// Mitsubishi GX Works2 project: RY300S2_3-4 24.07.21   PLC: Q03UDV
// RY300S2_3-4 24.07.21

PROGRAM MAIN
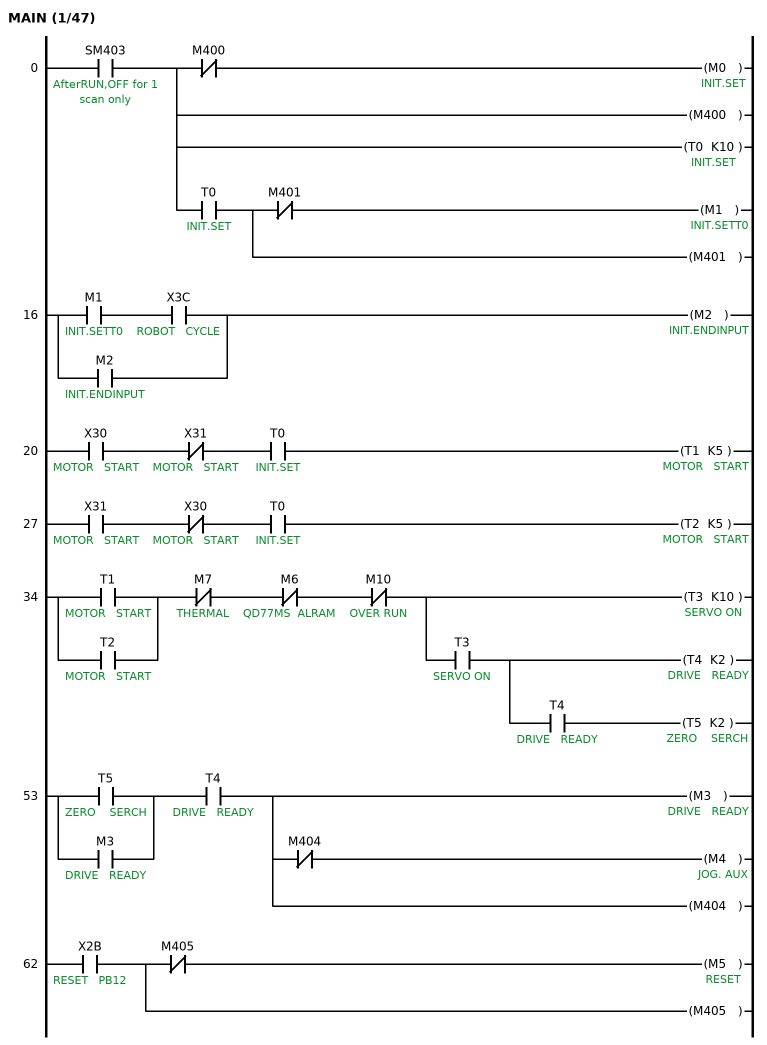
0     LD      SM403  ; AfterRUN,OFF for 1 scan only
      MPS
      ANI     M400
      OUT     M0  ; INIT.SET
      MPP
      OUT     M400
      OUT     T0 K10  ; INIT.SET
      AND     T0  ; INIT.SET
      MPS
      ANI     M401
      OUT     M1  ; INIT.SETT0
      MPP
      OUT     M401
16    LD      M1  ; INIT.SETT0
      AND     X3C  ; ROBOT   CYCLE
      OR      M2  ; INIT.ENDINPUT
      OUT     M2  ; INIT.ENDINPUT
20    LD      X30  ; MOTOR   START
      ANI     X31  ; MOTOR   START
      AND     T0  ; INIT.SET
      OUT     T1 K5  ; MOTOR   START
27    LD      X31  ; MOTOR   START
      ANI     X30  ; MOTOR   START
      AND     T0  ; INIT.SET
      OUT     T2 K5  ; MOTOR   START
34    LD      T1  ; MOTOR   START
      OR      T2  ; MOTOR   START
      ANI     M7  ; THERMAL
      ANI     M6  ; QD77MS  ALRAM
      ANI     M10  ; OVER RUN
      OUT     T3 K10  ; SERVO ON
      AND     T3  ; SERVO ON
      OUT     T4 K2  ; DRIVE   READY
      AND     T4  ; DRIVE   READY
      OUT     T5 K2  ; ZERO    SERCH
53    LD      T5  ; ZERO    SERCH
      OR      M3  ; DRIVE   READY
      AND     T4  ; DRIVE   READY
      OUT     M3  ; DRIVE   READY
      MPS
      ANI     M404
      OUT     M4  ; JOG. AUX
      MPP
      OUT     M404
62    LD      X2B  ; RESET   PB12
      MPS
      ANI     M405
      OUT     M5  ; RESET
      MPP
      OUT     M405
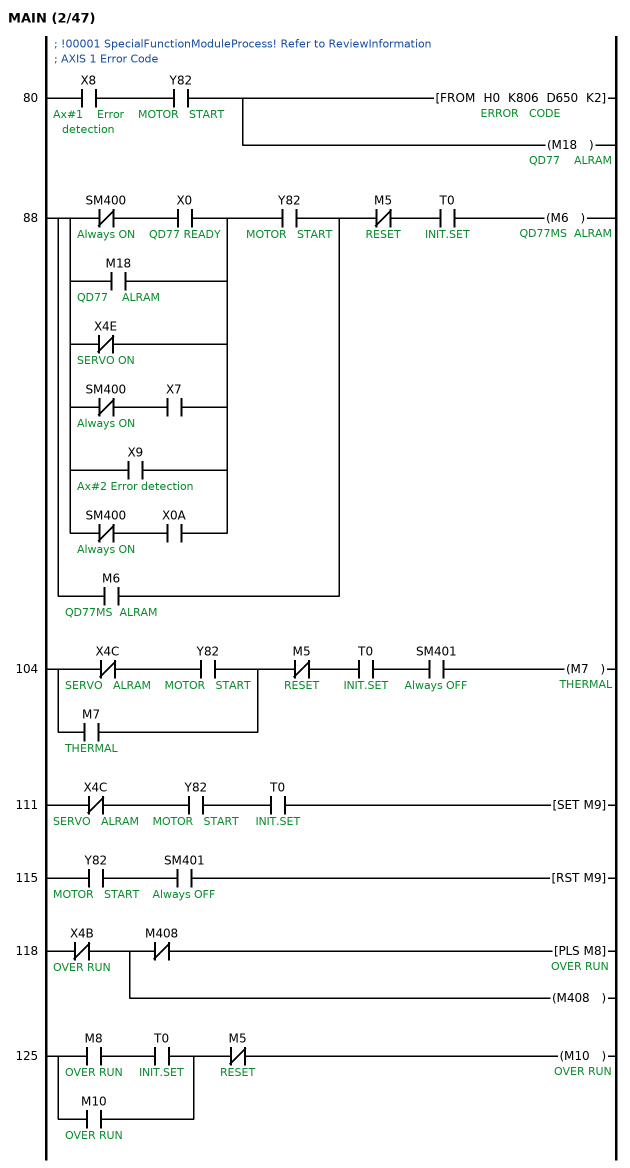
; !00001 SpecialFunctionModuleProcess! Refer to ReviewInformation
; AXIS 1 Error Code
80    LD      X8  ; Ax#1    Error   detection
      AND     Y82  ; MOTOR   START
      FROM    H0 K806 D650 K2  ; ERROR   CODE
      OUT     M18  ; QD77    ALRAM
88    LDI     SM400  ; Always ON
      AND     X0  ; QD77 READY
      OR      M18  ; QD77    ALRAM
      ORI     X4E  ; SERVO ON
      LDI     SM400  ; Always ON
      AND     X7
      ORB
      OR      X9  ; Ax#2 Error detection
      LDI     SM400  ; Always ON
      AND     X0A
      ORB
      AND     Y82  ; MOTOR   START
      OR      M6  ; QD77MS  ALRAM
      ANI     M5  ; RESET
      AND     T0  ; INIT.SET
      OUT     M6  ; QD77MS  ALRAM
104   LDI     X4C  ; SERVO   ALRAM
      AND     Y82  ; MOTOR   START
      OR      M7  ; THERMAL
      ANI     M5  ; RESET
      AND     T0  ; INIT.SET
      AND     SM401  ; Always OFF
      OUT     M7  ; THERMAL
111   LDI     X4C  ; SERVO   ALRAM
      AND     Y82  ; MOTOR   START
      AND     T0  ; INIT.SET
      SET     M9
115   LD      Y82  ; MOTOR   START
      AND     SM401  ; Always OFF
      RST     M9
118   LDI     X4B  ; OVER RUN
      MPS
      ANI     M408
      PLS     M8  ; OVER RUN
      MPP
      OUT     M408
125   LD      M8  ; OVER RUN
      AND     T0  ; INIT.SET
      OR      M10  ; OVER RUN
      ANI     M5  ; RESET
      OUT     M10  ; OVER RUN
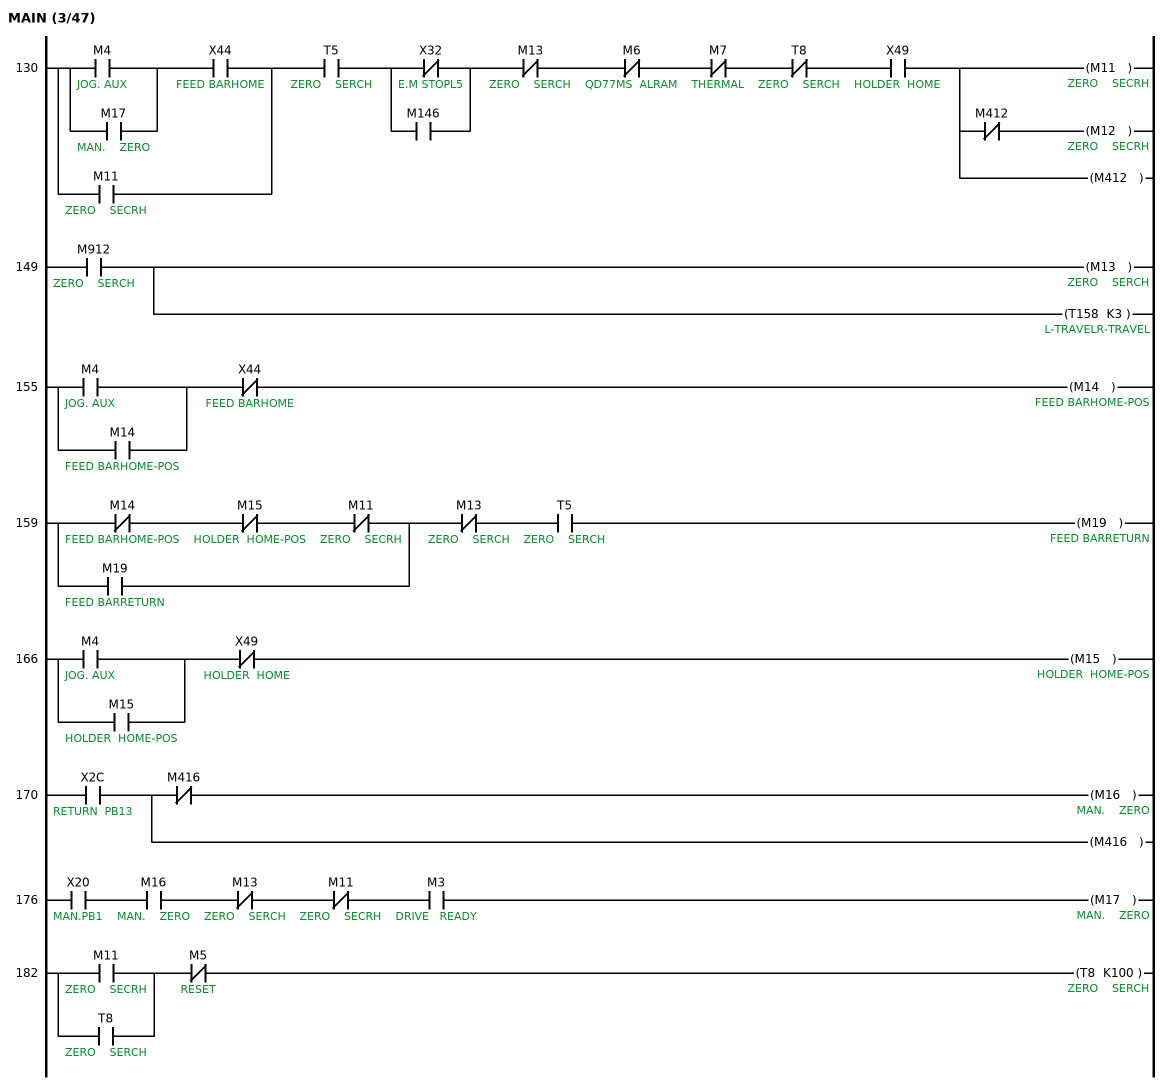
130   LD      M4  ; JOG. AUX
      OR      M17  ; MAN.    ZERO
      AND     X44  ; FEED BARHOME
      OR      M11  ; ZERO    SECRH
      AND     T5  ; ZERO    SERCH
      LDI     X32  ; E.M STOPL5
      OR      M146
      ANB
      ANI     M13  ; ZERO    SERCH
      ANI     M6  ; QD77MS  ALRAM
      ANI     M7  ; THERMAL
      ANI     T8  ; ZERO    SERCH
      AND     X49  ; HOLDER  HOME
      OUT     M11  ; ZERO    SECRH
      MPS
      ANI     M412
      OUT     M12  ; ZERO    SECRH
      MPP
      OUT     M412
149   LD      M912  ; ZERO    SERCH
      OUT     M13  ; ZERO    SERCH
      OUT     T158 K3  ; L-TRAVELR-TRAVEL
155   LD      M4  ; JOG. AUX
      OR      M14  ; FEED BARHOME-POS
      ANI     X44  ; FEED BARHOME
      OUT     M14  ; FEED BARHOME-POS
159   LDI     M14  ; FEED BARHOME-POS
      ANI     M15  ; HOLDER  HOME-POS
      ANI     M11  ; ZERO    SECRH
      OR      M19  ; FEED BARRETURN
      ANI     M13  ; ZERO    SERCH
      AND     T5  ; ZERO    SERCH
      OUT     M19  ; FEED BARRETURN
166   LD      M4  ; JOG. AUX
      OR      M15  ; HOLDER  HOME-POS
      ANI     X49  ; HOLDER  HOME
      OUT     M15  ; HOLDER  HOME-POS
170   LD      X2C  ; RETURN  PB13
      MPS
      ANI     M416
      OUT     M16  ; MAN.    ZERO
      MPP
      OUT     M416
176   LD      X20  ; MAN.PB1
      AND     M16  ; MAN.    ZERO
      ANI     M13  ; ZERO    SERCH
      ANI     M11  ; ZERO    SECRH
      AND     M3  ; DRIVE   READY
      OUT     M17  ; MAN.    ZERO
182   LD      M11  ; ZERO    SECRH
      OR      T8  ; ZERO    SERCH
      ANI     M5  ; RESET
      OUT     T8 K100  ; ZERO    SERCH
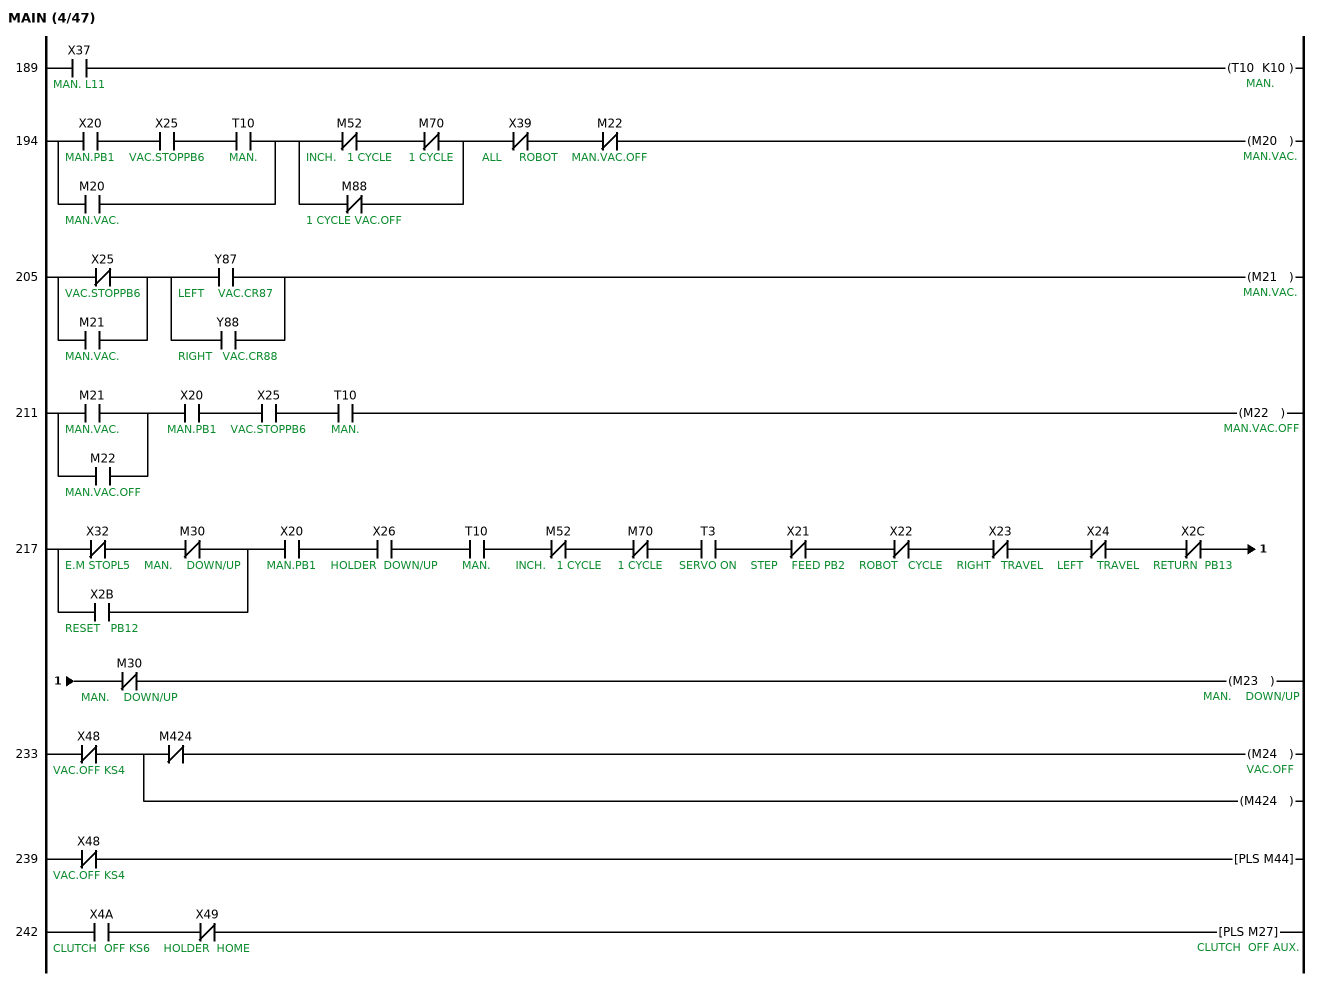
189   LD      X37  ; MAN. L11
      OUT     T10 K10  ; MAN.
194   LD      X20  ; MAN.PB1
      AND     X25  ; VAC.STOPPB6
      AND     T10  ; MAN.
      OR      M20  ; MAN.VAC.
      LDI     M52  ; INCH.   1 CYCLE
      ANI     M70  ; 1 CYCLE
      ORI     M88  ; 1 CYCLE VAC.OFF
      ANB
      ANI     X39  ; ALL     ROBOT
      ANI     M22  ; MAN.VAC.OFF
      OUT     M20  ; MAN.VAC.
205   LDI     X25  ; VAC.STOPPB6
      OR      M21  ; MAN.VAC.
      LD      Y87  ; LEFT    VAC.CR87
      OR      Y88  ; RIGHT   VAC.CR88
      ANB
      OUT     M21  ; MAN.VAC.
211   LD      M21  ; MAN.VAC.
      OR      M22  ; MAN.VAC.OFF
      AND     X20  ; MAN.PB1
      AND     X25  ; VAC.STOPPB6
      AND     T10  ; MAN.
      OUT     M22  ; MAN.VAC.OFF
217   LDI     X32  ; E.M STOPL5
      ANI     M30  ; MAN.    DOWN/UP
      OR      X2B  ; RESET   PB12
      AND     X20  ; MAN.PB1
      AND     X26  ; HOLDER  DOWN/UP
      AND     T10  ; MAN.
      ANI     M52  ; INCH.   1 CYCLE
      ANI     M70  ; 1 CYCLE
      AND     T3  ; SERVO ON
      ANI     X21  ; STEP    FEED PB2
      ANI     X22  ; ROBOT   CYCLE
      ANI     X23  ; RIGHT   TRAVEL
      ANI     X24  ; LEFT    TRAVEL
      ANI     X2C  ; RETURN  PB13
      ANI     M30  ; MAN.    DOWN/UP
      OUT     M23  ; MAN.    DOWN/UP
233   LDI     X48  ; VAC.OFF KS4
      MPS
      ANI     M424
      OUT     M24  ; VAC.OFF
      MPP
      OUT     M424
239   LDI     X48  ; VAC.OFF KS4
      PLS     M44
242   LD      X4A  ; CLUTCH  OFF KS6
      ANI     X49  ; HOLDER  HOME
      PLS     M27  ; CLUTCH  OFF AUX.
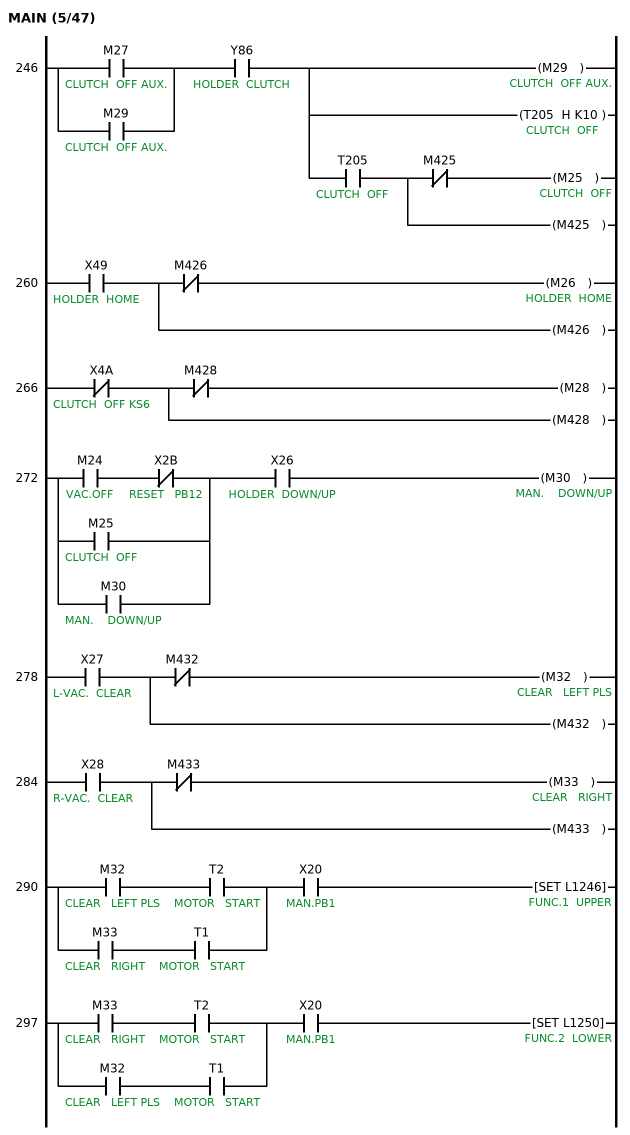
246   LD      M27  ; CLUTCH  OFF AUX.
      OR      M29  ; CLUTCH  OFF AUX.
      AND     Y86  ; HOLDER  CLUTCH
      OUT     M29  ; CLUTCH  OFF AUX.
      OUTH    T205 K10  ; CLUTCH  OFF
      AND     T205  ; CLUTCH  OFF
      MPS
      ANI     M425
      OUT     M25  ; CLUTCH  OFF
      MPP
      OUT     M425
260   LD      X49  ; HOLDER  HOME
      MPS
      ANI     M426
      OUT     M26  ; HOLDER  HOME
      MPP
      OUT     M426
266   LDI     X4A  ; CLUTCH  OFF KS6
      MPS
      ANI     M428
      OUT     M28
      MPP
      OUT     M428
272   LD      M24  ; VAC.OFF
      ANI     X2B  ; RESET   PB12
      OR      M25  ; CLUTCH  OFF
      OR      M30  ; MAN.    DOWN/UP
      AND     X26  ; HOLDER  DOWN/UP
      OUT     M30  ; MAN.    DOWN/UP
278   LD      X27  ; L-VAC.  CLEAR
      MPS
      ANI     M432
      OUT     M32  ; CLEAR   LEFT PLS
      MPP
      OUT     M432
284   LD      X28  ; R-VAC.  CLEAR
      MPS
      ANI     M433
      OUT     M33  ; CLEAR   RIGHT
      MPP
      OUT     M433
290   LD      M32  ; CLEAR   LEFT PLS
      AND     T2  ; MOTOR   START
      LD      M33  ; CLEAR   RIGHT
      AND     T1  ; MOTOR   START
      ORB
      AND     X20  ; MAN.PB1
      SET     L1246  ; FUNC.1  UPPER
297   LD      M33  ; CLEAR   RIGHT
      AND     T2  ; MOTOR   START
      LD      M32  ; CLEAR   LEFT PLS
      AND     T1  ; MOTOR   START
      ORB
      AND     X20  ; MAN.PB1
      SET     L1250  ; FUNC.2  LOWER
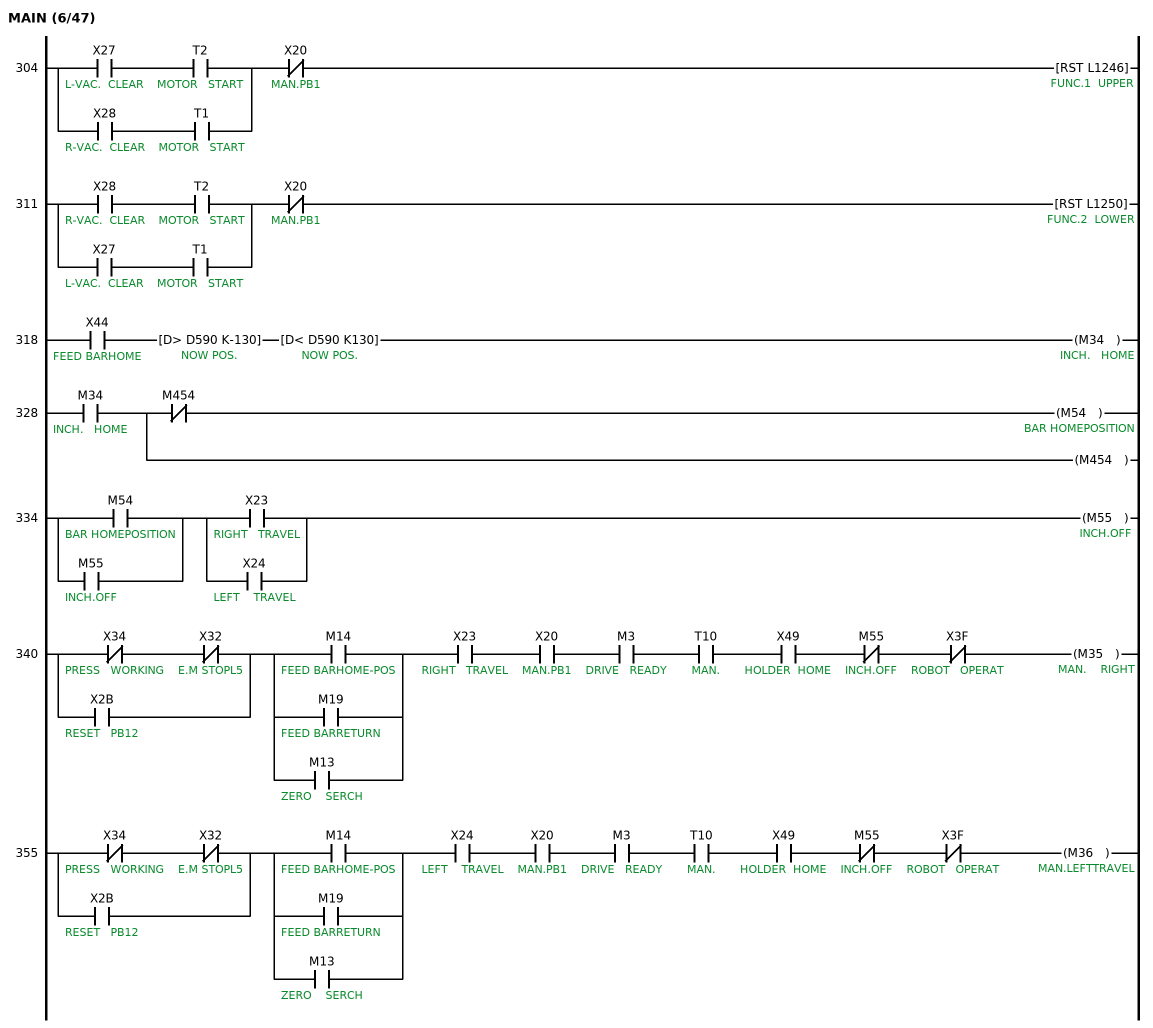
304   LD      X27  ; L-VAC.  CLEAR
      AND     T2  ; MOTOR   START
      LD      X28  ; R-VAC.  CLEAR
      AND     T1  ; MOTOR   START
      ORB
      ANI     X20  ; MAN.PB1
      RST     L1246  ; FUNC.1  UPPER
311   LD      X28  ; R-VAC.  CLEAR
      AND     T2  ; MOTOR   START
      LD      X27  ; L-VAC.  CLEAR
      AND     T1  ; MOTOR   START
      ORB
      ANI     X20  ; MAN.PB1
      RST     L1250  ; FUNC.2  LOWER
318   LD      X44  ; FEED BARHOME
      ANDD>   D590 K-130  ; NOW POS.
      ANDD<   D590 K130  ; NOW POS.
      OUT     M34  ; INCH.   HOME
328   LD      M34  ; INCH.   HOME
      MPS
      ANI     M454
      OUT     M54  ; BAR HOMEPOSITION
      MPP
      OUT     M454
334   LD      M54  ; BAR HOMEPOSITION
      OR      M55  ; INCH.OFF
      LD      X23  ; RIGHT   TRAVEL
      OR      X24  ; LEFT    TRAVEL
      ANB
      OUT     M55  ; INCH.OFF
340   LDI     X34  ; PRESS   WORKING
      ANI     X32  ; E.M STOPL5
      OR      X2B  ; RESET   PB12
      LD      M14  ; FEED BARHOME-POS
      OR      M19  ; FEED BARRETURN
      OR      M13  ; ZERO    SERCH
      ANB
      AND     X23  ; RIGHT   TRAVEL
      AND     X20  ; MAN.PB1
      AND     M3  ; DRIVE   READY
      AND     T10  ; MAN.
      AND     X49  ; HOLDER  HOME
      ANI     M55  ; INCH.OFF
      ANI     X3F  ; ROBOT   OPERAT
      OUT     M35  ; MAN.    RIGHT
355   LDI     X34  ; PRESS   WORKING
      ANI     X32  ; E.M STOPL5
      OR      X2B  ; RESET   PB12
      LD      M14  ; FEED BARHOME-POS
      OR      M19  ; FEED BARRETURN
      OR      M13  ; ZERO    SERCH
      ANB
      AND     X24  ; LEFT    TRAVEL
      AND     X20  ; MAN.PB1
      AND     M3  ; DRIVE   READY
      AND     T10  ; MAN.
      AND     X49  ; HOLDER  HOME
      ANI     M55  ; INCH.OFF
      ANI     X3F  ; ROBOT   OPERAT
      OUT     M36  ; MAN.LEFTTRAVEL
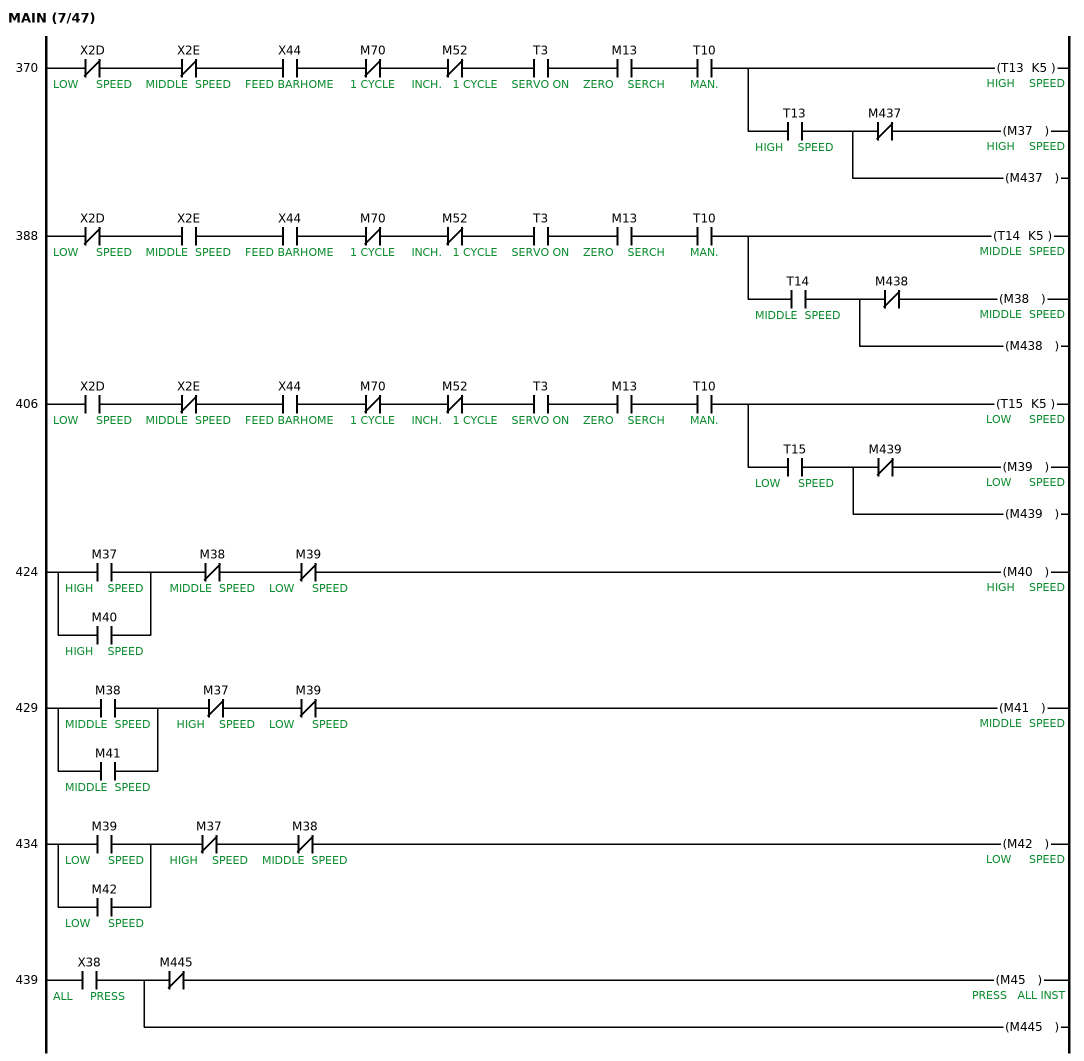
370   LDI     X2D  ; LOW     SPEED
      ANI     X2E  ; MIDDLE  SPEED
      AND     X44  ; FEED BARHOME
      ANI     M70  ; 1 CYCLE
      ANI     M52  ; INCH.   1 CYCLE
      AND     T3  ; SERVO ON
      AND     M13  ; ZERO    SERCH
      AND     T10  ; MAN.
      OUT     T13 K5  ; HIGH    SPEED
      AND     T13  ; HIGH    SPEED
      MPS
      ANI     M437
      OUT     M37  ; HIGH    SPEED
      MPP
      OUT     M437
388   LDI     X2D  ; LOW     SPEED
      AND     X2E  ; MIDDLE  SPEED
      AND     X44  ; FEED BARHOME
      ANI     M70  ; 1 CYCLE
      ANI     M52  ; INCH.   1 CYCLE
      AND     T3  ; SERVO ON
      AND     M13  ; ZERO    SERCH
      AND     T10  ; MAN.
      OUT     T14 K5  ; MIDDLE  SPEED
      AND     T14  ; MIDDLE  SPEED
      MPS
      ANI     M438
      OUT     M38  ; MIDDLE  SPEED
      MPP
      OUT     M438
406   LD      X2D  ; LOW     SPEED
      ANI     X2E  ; MIDDLE  SPEED
      AND     X44  ; FEED BARHOME
      ANI     M70  ; 1 CYCLE
      ANI     M52  ; INCH.   1 CYCLE
      AND     T3  ; SERVO ON
      AND     M13  ; ZERO    SERCH
      AND     T10  ; MAN.
      OUT     T15 K5  ; LOW     SPEED
      AND     T15  ; LOW     SPEED
      MPS
      ANI     M439
      OUT     M39  ; LOW     SPEED
      MPP
      OUT     M439
424   LD      M37  ; HIGH    SPEED
      OR      M40  ; HIGH    SPEED
      ANI     M38  ; MIDDLE  SPEED
      ANI     M39  ; LOW     SPEED
      OUT     M40  ; HIGH    SPEED
429   LD      M38  ; MIDDLE  SPEED
      OR      M41  ; MIDDLE  SPEED
      ANI     M37  ; HIGH    SPEED
      ANI     M39  ; LOW     SPEED
      OUT     M41  ; MIDDLE  SPEED
434   LD      M39  ; LOW     SPEED
      OR      M42  ; LOW     SPEED
      ANI     M37  ; HIGH    SPEED
      ANI     M38  ; MIDDLE  SPEED
      OUT     M42  ; LOW     SPEED
439   LD      X38  ; ALL     PRESS
      MPS
      ANI     M445
      OUT     M45  ; PRESS   ALL INST
      MPP
      OUT     M445
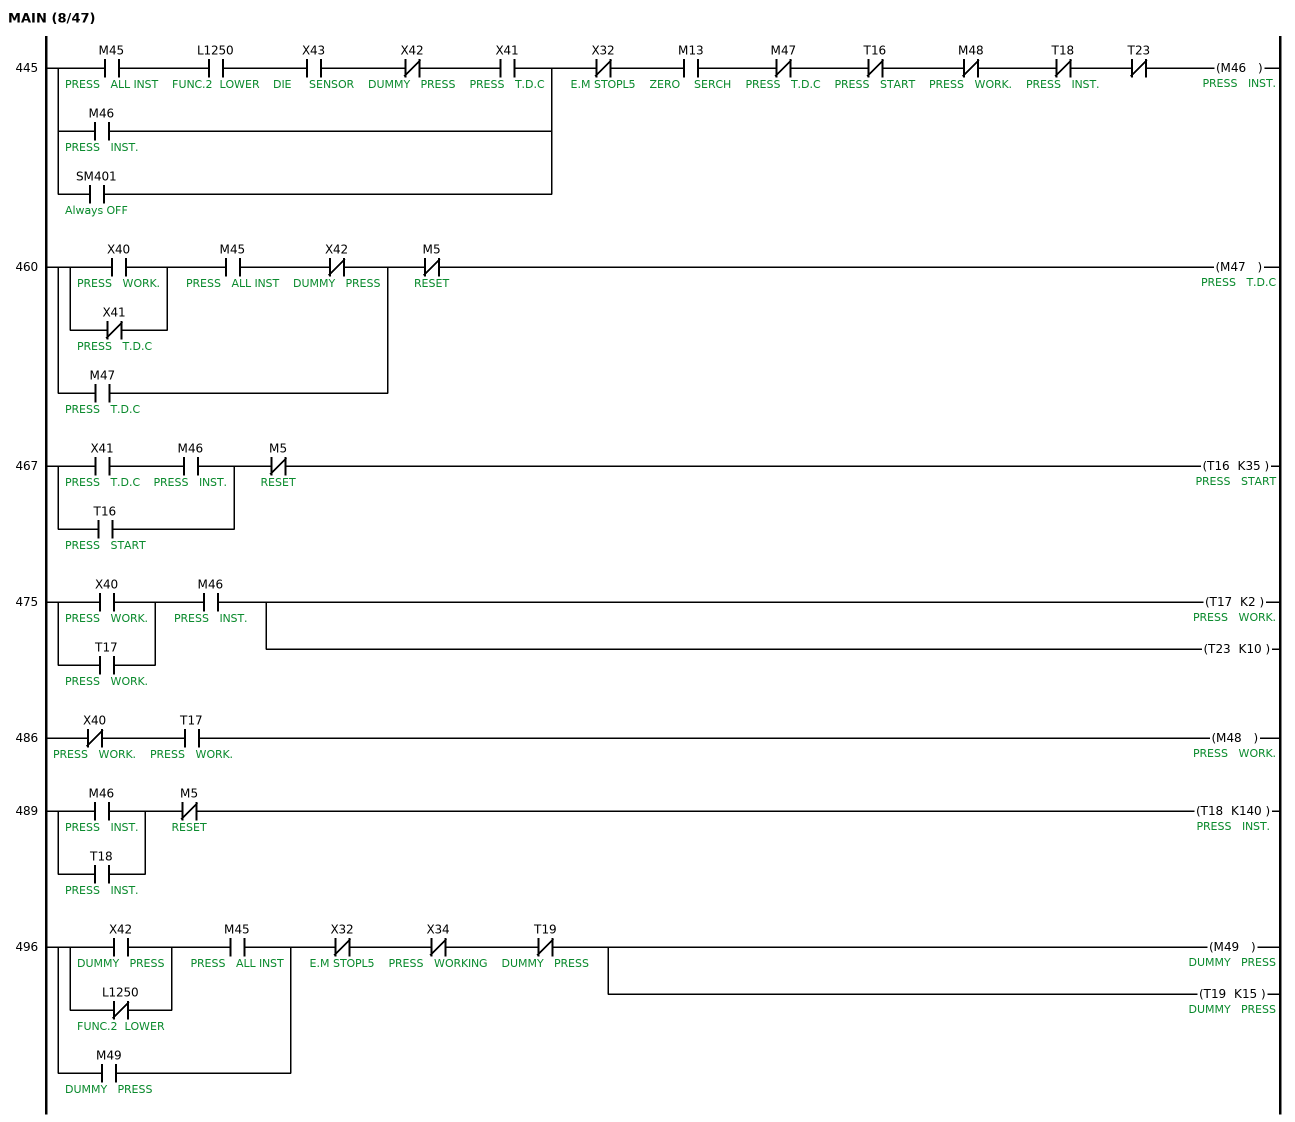
445   LD      M45  ; PRESS   ALL INST
      AND     L1250  ; FUNC.2  LOWER
      AND     X43  ; DIE     SENSOR
      ANI     X42  ; DUMMY   PRESS
      AND     X41  ; PRESS   T.D.C
      OR      M46  ; PRESS   INST.
      OR      SM401  ; Always OFF
      ANI     X32  ; E.M STOPL5
      AND     M13  ; ZERO    SERCH
      ANI     M47  ; PRESS   T.D.C
      ANI     T16  ; PRESS   START
      ANI     M48  ; PRESS   WORK.
      ANI     T18  ; PRESS   INST.
      ANI     T23
      OUT     M46  ; PRESS   INST.
460   LD      X40  ; PRESS   WORK.
      ORI     X41  ; PRESS   T.D.C
      AND     M45  ; PRESS   ALL INST
      ANI     X42  ; DUMMY   PRESS
      OR      M47  ; PRESS   T.D.C
      ANI     M5  ; RESET
      OUT     M47  ; PRESS   T.D.C
467   LD      X41  ; PRESS   T.D.C
      AND     M46  ; PRESS   INST.
      OR      T16  ; PRESS   START
      ANI     M5  ; RESET
      OUT     T16 K35  ; PRESS   START
475   LD      X40  ; PRESS   WORK.
      OR      T17  ; PRESS   WORK.
      AND     M46  ; PRESS   INST.
      OUT     T17 K2  ; PRESS   WORK.
      OUT     T23 K10
486   LDI     X40  ; PRESS   WORK.
      AND     T17  ; PRESS   WORK.
      OUT     M48  ; PRESS   WORK.
489   LD      M46  ; PRESS   INST.
      OR      T18  ; PRESS   INST.
      ANI     M5  ; RESET
      OUT     T18 K140  ; PRESS   INST.
496   LD      X42  ; DUMMY   PRESS
      ORI     L1250  ; FUNC.2  LOWER
      AND     M45  ; PRESS   ALL INST
      OR      M49  ; DUMMY   PRESS
      ANI     X32  ; E.M STOPL5
      ANI     X34  ; PRESS   WORKING
      ANI     T19  ; DUMMY   PRESS
      OUT     M49  ; DUMMY   PRESS
      OUT     T19 K15  ; DUMMY   PRESS
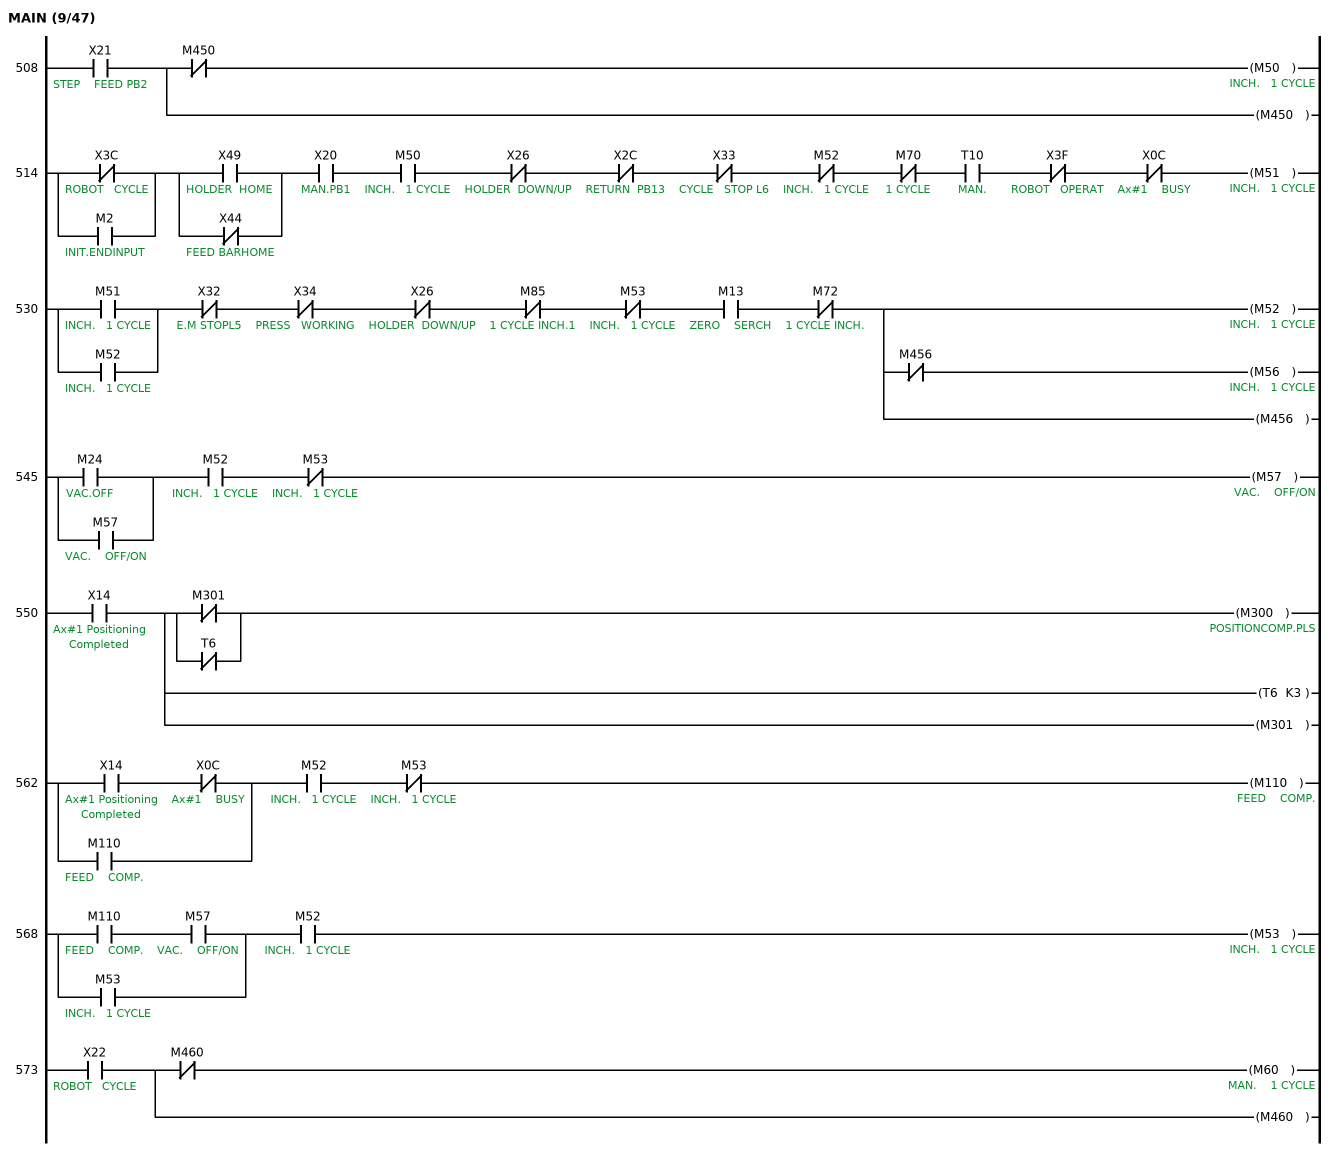
508   LD      X21  ; STEP    FEED PB2
      MPS
      ANI     M450
      OUT     M50  ; INCH.   1 CYCLE
      MPP
      OUT     M450
514   LDI     X3C  ; ROBOT   CYCLE
      OR      M2  ; INIT.ENDINPUT
      LD      X49  ; HOLDER  HOME
      ORI     X44  ; FEED BARHOME
      ANB
      AND     X20  ; MAN.PB1
      AND     M50  ; INCH.   1 CYCLE
      ANI     X26  ; HOLDER  DOWN/UP
      ANI     X2C  ; RETURN  PB13
      ANI     X33  ; CYCLE   STOP L6
      ANI     M52  ; INCH.   1 CYCLE
      ANI     M70  ; 1 CYCLE
      AND     T10  ; MAN.
      ANI     X3F  ; ROBOT   OPERAT
      ANI     X0C  ; Ax#1    BUSY
      OUT     M51  ; INCH.   1 CYCLE
530   LD      M51  ; INCH.   1 CYCLE
      OR      M52  ; INCH.   1 CYCLE
      ANI     X32  ; E.M STOPL5
      ANI     X34  ; PRESS   WORKING
      ANI     X26  ; HOLDER  DOWN/UP
      ANI     M85  ; 1 CYCLE INCH.1
      ANI     M53  ; INCH.   1 CYCLE
      AND     M13  ; ZERO    SERCH
      ANI     M72  ; 1 CYCLE INCH.
      OUT     M52  ; INCH.   1 CYCLE
      MPS
      ANI     M456
      OUT     M56  ; INCH.   1 CYCLE
      MPP
      OUT     M456
545   LD      M24  ; VAC.OFF
      OR      M57  ; VAC.    OFF/ON
      AND     M52  ; INCH.   1 CYCLE
      ANI     M53  ; INCH.   1 CYCLE
      OUT     M57  ; VAC.    OFF/ON
550   LD      X14  ; Ax#1 PositioningCompleted
      MPS
      LDI     M301
      ORI     T6
      ANB
      OUT     M300  ; POSITIONCOMP.PLS
      MPP
      OUT     T6 K3
      OUT     M301
562   LD      X14  ; Ax#1 PositioningCompleted
      ANI     X0C  ; Ax#1    BUSY
      OR      M110  ; FEED    COMP.
      AND     M52  ; INCH.   1 CYCLE
      ANI     M53  ; INCH.   1 CYCLE
      OUT     M110  ; FEED    COMP.
568   LD      M110  ; FEED    COMP.
      AND     M57  ; VAC.    OFF/ON
      OR      M53  ; INCH.   1 CYCLE
      AND     M52  ; INCH.   1 CYCLE
      OUT     M53  ; INCH.   1 CYCLE
573   LD      X22  ; ROBOT   CYCLE
      MPS
      ANI     M460
      OUT     M60  ; MAN.    1 CYCLE
      MPP
      OUT     M460
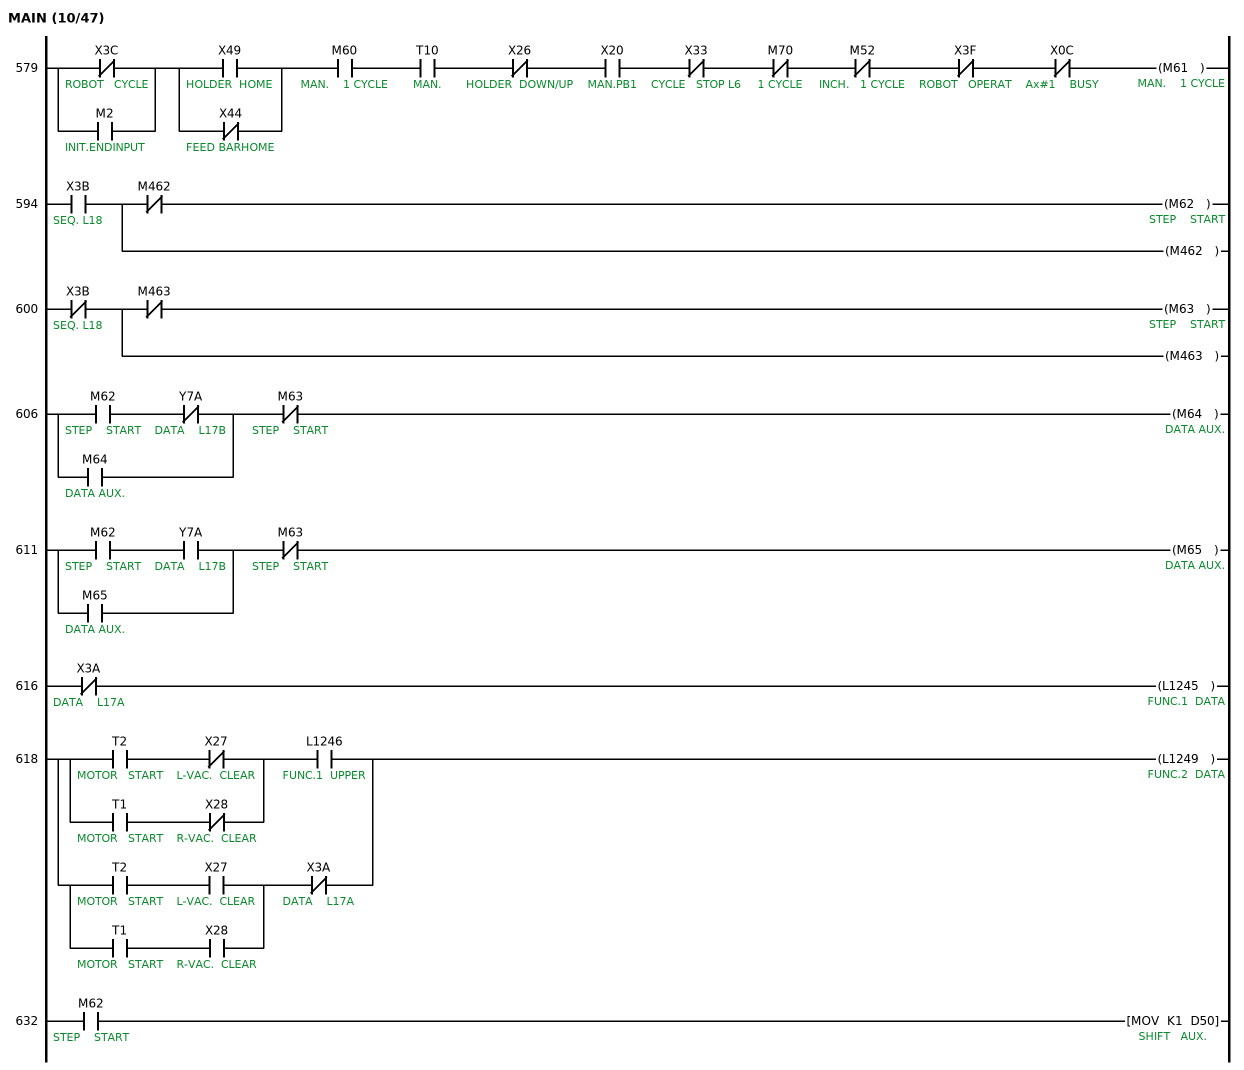
579   LDI     X3C  ; ROBOT   CYCLE
      OR      M2  ; INIT.ENDINPUT
      LD      X49  ; HOLDER  HOME
      ORI     X44  ; FEED BARHOME
      ANB
      AND     M60  ; MAN.    1 CYCLE
      AND     T10  ; MAN.
      ANI     X26  ; HOLDER  DOWN/UP
      AND     X20  ; MAN.PB1
      ANI     X33  ; CYCLE   STOP L6
      ANI     M70  ; 1 CYCLE
      ANI     M52  ; INCH.   1 CYCLE
      ANI     X3F  ; ROBOT   OPERAT
      ANI     X0C  ; Ax#1    BUSY
      OUT     M61  ; MAN.    1 CYCLE
594   LD      X3B  ; SEQ. L18
      MPS
      ANI     M462
      OUT     M62  ; STEP    START
      MPP
      OUT     M462
600   LDI     X3B  ; SEQ. L18
      MPS
      ANI     M463
      OUT     M63  ; STEP    START
      MPP
      OUT     M463
606   LD      M62  ; STEP    START
      ANI     Y7A  ; DATA    L17B
      OR      M64  ; DATA AUX.
      ANI     M63  ; STEP    START
      OUT     M64  ; DATA AUX.
611   LD      M62  ; STEP    START
      AND     Y7A  ; DATA    L17B
      OR      M65  ; DATA AUX.
      ANI     M63  ; STEP    START
      OUT     M65  ; DATA AUX.
616   LDI     X3A  ; DATA    L17A
      OUT     L1245  ; FUNC.1  DATA
618   LD      T2  ; MOTOR   START
      ANI     X27  ; L-VAC.  CLEAR
      LD      T1  ; MOTOR   START
      ANI     X28  ; R-VAC.  CLEAR
      ORB
      AND     L1246  ; FUNC.1  UPPER
      LD      T2  ; MOTOR   START
      AND     X27  ; L-VAC.  CLEAR
      LD      T1  ; MOTOR   START
      AND     X28  ; R-VAC.  CLEAR
      ORB
      ANI     X3A  ; DATA    L17A
      ORB
      OUT     L1249  ; FUNC.2  DATA
632   LD      M62  ; STEP    START
      MOV     K1 D50  ; SHIFT   AUX.
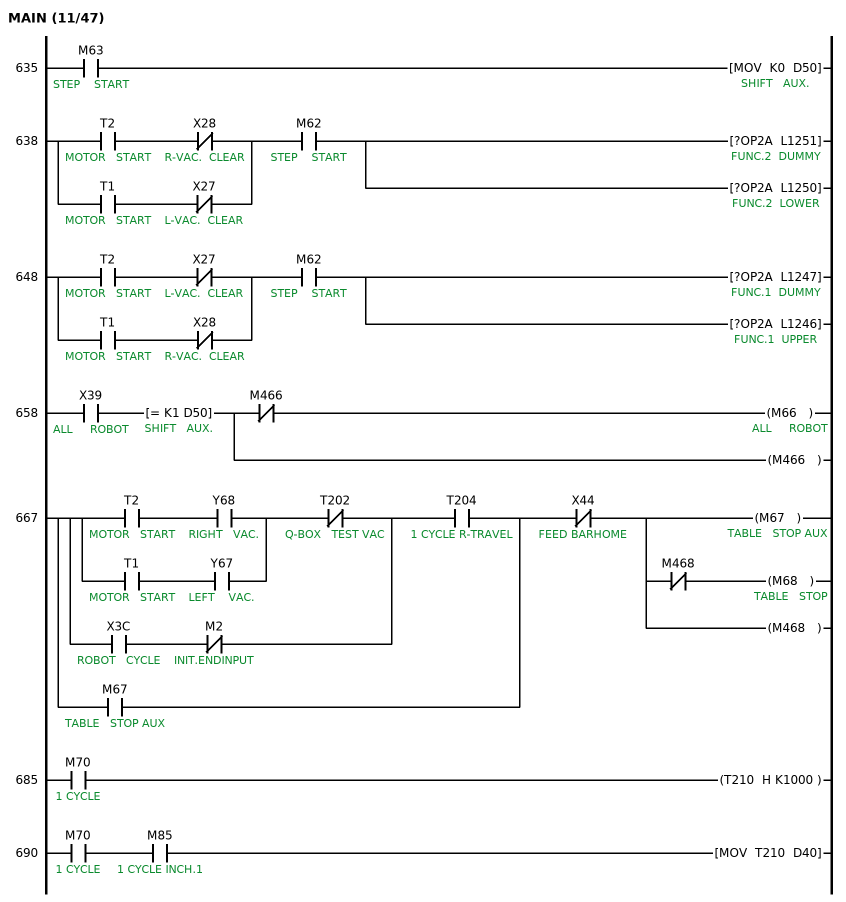
635   LD      M63  ; STEP    START
      MOV     K0 D50
638   LD      T2  ; MOTOR   START
      ANI     X28  ; R-VAC.  CLEAR
      LD      T1  ; MOTOR   START
      ANI     X27  ; L-VAC.  CLEAR
      ORB
      AND     M62  ; STEP    START
      ?OP2A   L1251  ; FUNC.2  DUMMY
      ?OP2A   L1250
648   LD      T2  ; MOTOR   START
      ANI     X27  ; L-VAC.  CLEAR
      LD      T1  ; MOTOR   START
      ANI     X28  ; R-VAC.  CLEAR
      ORB
      AND     M62  ; STEP    START
      ?OP2A   L1247  ; FUNC.1  DUMMY
      ?OP2A   L1246
658   LD      X39  ; ALL     ROBOT
      AND=    K1 D50  ; SHIFT   AUX.
      MPS
      ANI     M466
      OUT     M66  ; ALL     ROBOT
      MPP
      OUT     M466
667   LD      T2  ; MOTOR   START
      AND     Y68  ; RIGHT   VAC.
      LD      T1  ; MOTOR   START
      AND     Y67  ; LEFT    VAC.
      ORB
      ANI     T202  ; Q-BOX   TEST VAC
      LD      X3C  ; ROBOT   CYCLE
      ANI     M2  ; INIT.ENDINPUT
      ORB
      AND     T204  ; 1 CYCLE R-TRAVEL
      OR      M67  ; TABLE   STOP AUX
      ANI     X44  ; FEED BARHOME
      OUT     M67  ; TABLE   STOP AUX
      MPS
      ANI     M468
      OUT     M68  ; TABLE   STOP
      MPP
      OUT     M468
685   LD      M70  ; 1 CYCLE
      OUTH    T210 K1000
690   LD      M70  ; 1 CYCLE
      AND     M85  ; 1 CYCLE INCH.1
      MOV     T210 D40
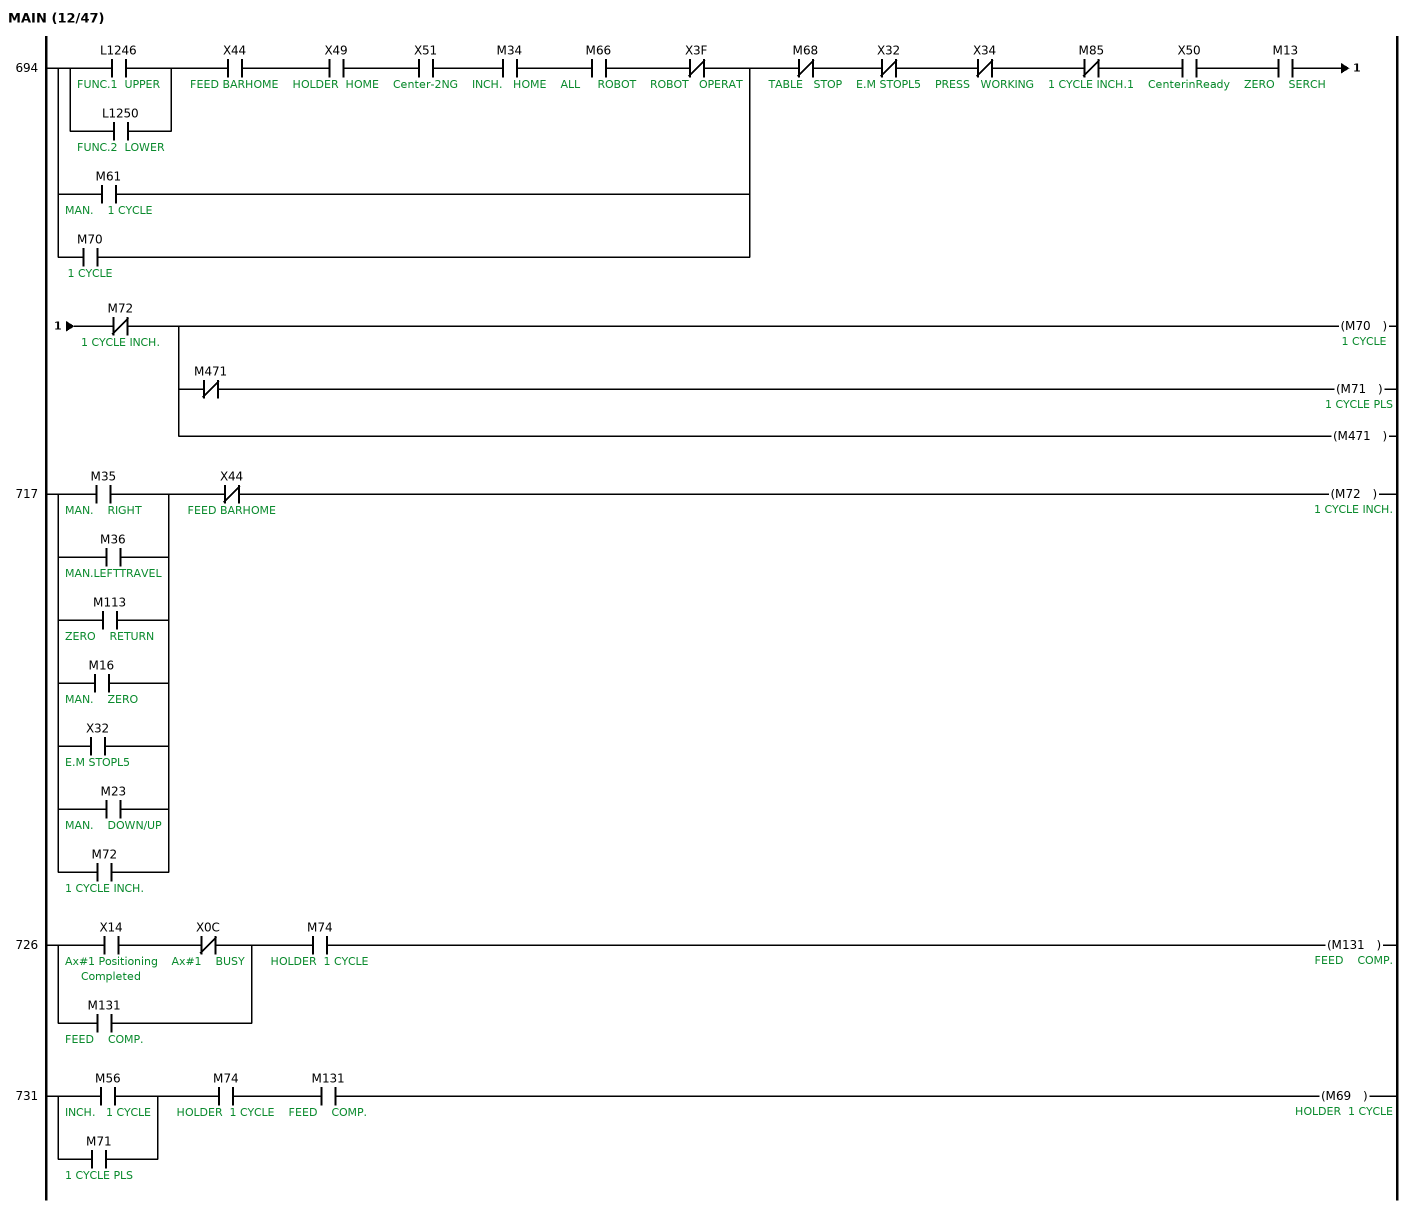
694   LD      L1246  ; FUNC.1  UPPER
      OR      L1250  ; FUNC.2  LOWER
      AND     X44  ; FEED BARHOME
      AND     X49  ; HOLDER  HOME
      AND     X51  ; Center-2NG
      AND     M34  ; INCH.   HOME
      AND     M66  ; ALL     ROBOT
      ANI     X3F  ; ROBOT   OPERAT
      OR      M61  ; MAN.    1 CYCLE
      OR      M70  ; 1 CYCLE
      ANI     M68  ; TABLE   STOP
      ANI     X32  ; E.M STOPL5
      ANI     X34  ; PRESS   WORKING
      ANI     M85  ; 1 CYCLE INCH.1
      AND     X50  ; CenterinReady
      AND     M13  ; ZERO    SERCH
      ANI     M72  ; 1 CYCLE INCH.
      OUT     M70  ; 1 CYCLE
      MPS
      ANI     M471
      OUT     M71  ; 1 CYCLE PLS
      MPP
      OUT     M471
717   LD      M35  ; MAN.    RIGHT
      OR      M36  ; MAN.LEFTTRAVEL
      OR      M113  ; ZERO    RETURN
      OR      M16  ; MAN.    ZERO
      OR      X32  ; E.M STOPL5
      OR      M23  ; MAN.    DOWN/UP
      OR      M72  ; 1 CYCLE INCH.
      ANI     X44  ; FEED BARHOME
      OUT     M72  ; 1 CYCLE INCH.
726   LD      X14  ; Ax#1 PositioningCompleted
      ANI     X0C  ; Ax#1    BUSY
      OR      M131  ; FEED    COMP.
      AND     M74  ; HOLDER  1 CYCLE
      OUT     M131  ; FEED    COMP.
731   LD      M56  ; INCH.   1 CYCLE
      OR      M71  ; 1 CYCLE PLS
      AND     M74  ; HOLDER  1 CYCLE
      AND     M131  ; FEED    COMP.
      OUT     M69  ; HOLDER  1 CYCLE
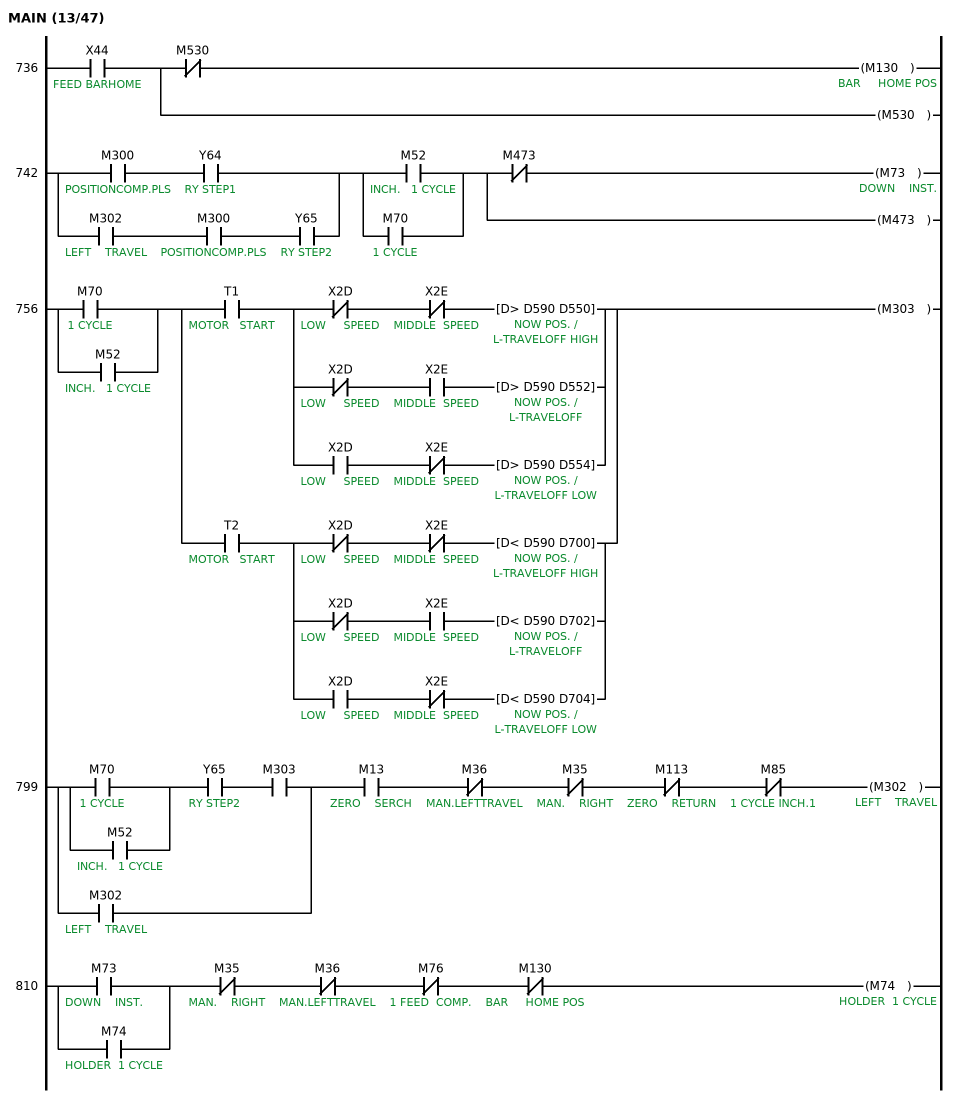
736   LD      X44  ; FEED BARHOME
      MPS
      ANI     M530
      OUT     M130  ; BAR     HOME POS
      MPP
      OUT     M530
742   LD      M300  ; POSITIONCOMP.PLS
      AND     Y64  ; RY STEP1
      LD      M302  ; LEFT    TRAVEL
      AND     M300  ; POSITIONCOMP.PLS
      AND     Y65  ; RY STEP2
      ORB
      LD      M52  ; INCH.   1 CYCLE
      OR      M70  ; 1 CYCLE
      ANB
      MPS
      ANI     M473
      OUT     M73  ; DOWN    INST.
      MPP
      OUT     M473
756   LD      M70  ; 1 CYCLE
      OR      M52  ; INCH.   1 CYCLE
      LD      T1  ; MOTOR   START
      LDI     X2D  ; LOW     SPEED
      ANI     X2E  ; MIDDLE  SPEED
      ANDD>   D590 D550  ; NOW POS. / L-TRAVELOFF HIGH
      LDI     X2D  ; LOW     SPEED
      AND     X2E  ; MIDDLE  SPEED
      ANDD>   D590 D552  ; NOW POS. / L-TRAVELOFF
      ORB
      LD      X2D  ; LOW     SPEED
      ANI     X2E  ; MIDDLE  SPEED
      ANDD>   D590 D554  ; NOW POS. / L-TRAVELOFF LOW
      ORB
      ANB
      LD      T2  ; MOTOR   START
      LDI     X2D  ; LOW     SPEED
      ANI     X2E  ; MIDDLE  SPEED
      ANDD<   D590 D700  ; NOW POS. / L-TRAVELOFF HIGH
      LDI     X2D  ; LOW     SPEED
      AND     X2E  ; MIDDLE  SPEED
      ANDD<   D590 D702  ; NOW POS. / L-TRAVELOFF
      ORB
      LD      X2D  ; LOW     SPEED
      ANI     X2E  ; MIDDLE  SPEED
      ANDD<   D590 D704  ; NOW POS. / L-TRAVELOFF LOW
      ORB
      ANB
      ORB
      ANB
      OUT     M303
799   LD      M70  ; 1 CYCLE
      OR      M52  ; INCH.   1 CYCLE
      AND     Y65  ; RY STEP2
      AND     M303
      OR      M302  ; LEFT    TRAVEL
      AND     M13  ; ZERO    SERCH
      ANI     M36  ; MAN.LEFTTRAVEL
      ANI     M35  ; MAN.    RIGHT
      ANI     M113  ; ZERO    RETURN
      ANI     M85  ; 1 CYCLE INCH.1
      OUT     M302  ; LEFT    TRAVEL
810   LD      M73  ; DOWN    INST.
      OR      M74  ; HOLDER  1 CYCLE
      ANI     M35  ; MAN.    RIGHT
      ANI     M36  ; MAN.LEFTTRAVEL
      ANI     M76  ; 1 FEED  COMP.
      ANI     M130  ; BAR     HOME POS
      OUT     M74  ; HOLDER  1 CYCLE
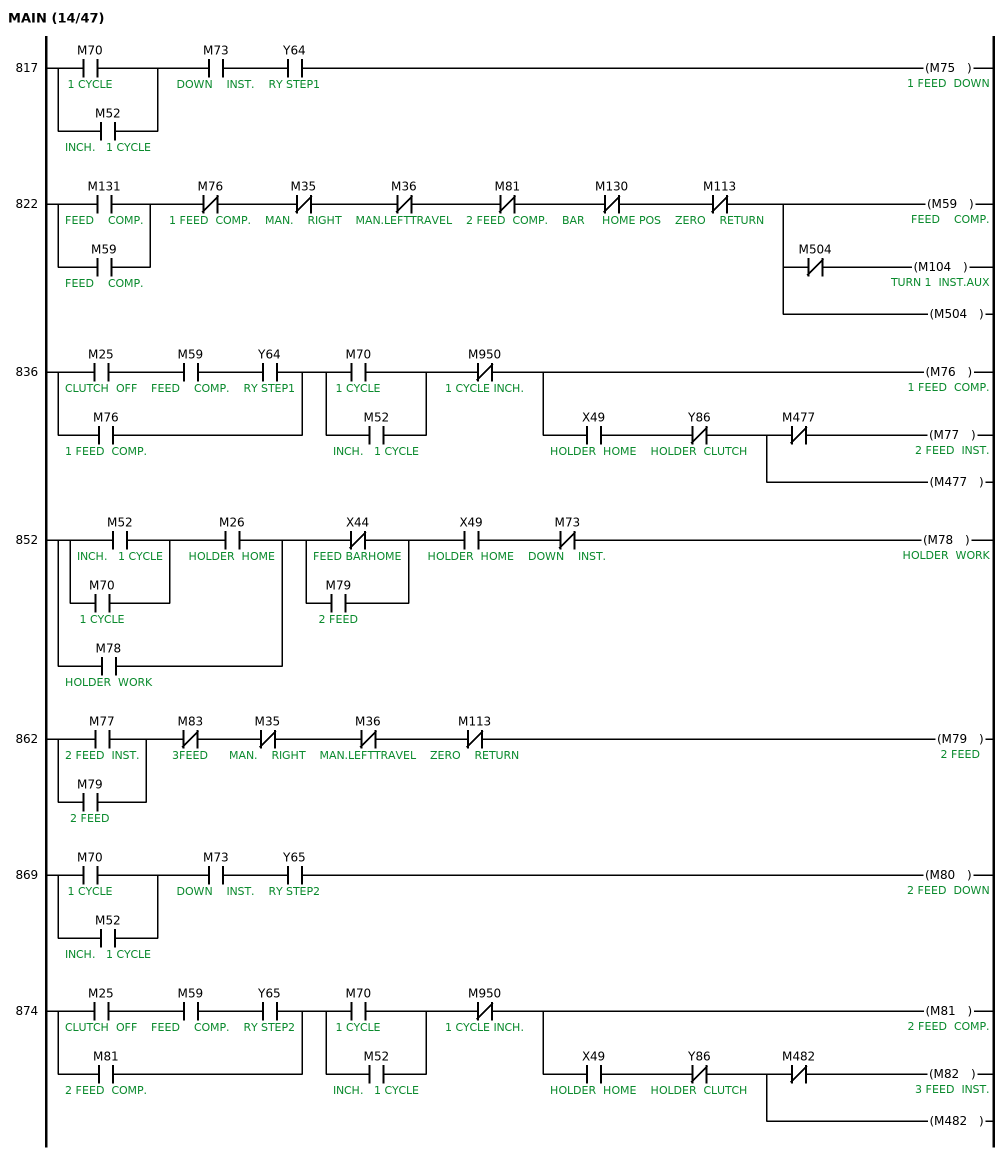
817   LD      M70  ; 1 CYCLE
      OR      M52  ; INCH.   1 CYCLE
      AND     M73  ; DOWN    INST.
      AND     Y64  ; RY STEP1
      OUT     M75  ; 1 FEED  DOWN
822   LD      M131  ; FEED    COMP.
      OR      M59  ; FEED    COMP.
      ANI     M76  ; 1 FEED  COMP.
      ANI     M35  ; MAN.    RIGHT
      ANI     M36  ; MAN.LEFTTRAVEL
      ANI     M81  ; 2 FEED  COMP.
      ANI     M130  ; BAR     HOME POS
      ANI     M113  ; ZERO    RETURN
      OUT     M59  ; FEED    COMP.
      MPS
      ANI     M504
      OUT     M104  ; TURN 1  INST.AUX
      MPP
      OUT     M504
836   LD      M25  ; CLUTCH  OFF
      AND     M59  ; FEED    COMP.
      AND     Y64  ; RY STEP1
      OR      M76  ; 1 FEED  COMP.
      LD      M70  ; 1 CYCLE
      OR      M52  ; INCH.   1 CYCLE
      ANB
      ANI     M950  ; 1 CYCLE INCH.
      OUT     M76  ; 1 FEED  COMP.
      AND     X49  ; HOLDER  HOME
      ANI     Y86  ; HOLDER  CLUTCH
      MPS
      ANI     M477
      OUT     M77  ; 2 FEED  INST.
      MPP
      OUT     M477
852   LD      M52  ; INCH.   1 CYCLE
      OR      M70  ; 1 CYCLE
      AND     M26  ; HOLDER  HOME
      OR      M78  ; HOLDER  WORK
      LDI     X44  ; FEED BARHOME
      OR      M79  ; 2 FEED
      ANB
      AND     X49  ; HOLDER  HOME
      ANI     M73  ; DOWN    INST.
      OUT     M78  ; HOLDER  WORK
862   LD      M77  ; 2 FEED  INST.
      OR      M79  ; 2 FEED
      ANI     M83  ; 3FEED
      ANI     M35  ; MAN.    RIGHT
      ANI     M36  ; MAN.LEFTTRAVEL
      ANI     M113  ; ZERO    RETURN
      OUT     M79  ; 2 FEED
869   LD      M70  ; 1 CYCLE
      OR      M52  ; INCH.   1 CYCLE
      AND     M73  ; DOWN    INST.
      AND     Y65  ; RY STEP2
      OUT     M80  ; 2 FEED  DOWN
874   LD      M25  ; CLUTCH  OFF
      AND     M59  ; FEED    COMP.
      AND     Y65  ; RY STEP2
      OR      M81  ; 2 FEED  COMP.
      LD      M70  ; 1 CYCLE
      OR      M52  ; INCH.   1 CYCLE
      ANB
      ANI     M950  ; 1 CYCLE INCH.
      OUT     M81  ; 2 FEED  COMP.
      AND     X49  ; HOLDER  HOME
      ANI     Y86  ; HOLDER  CLUTCH
      MPS
      ANI     M482
      OUT     M82  ; 3 FEED  INST.
      MPP
      OUT     M482
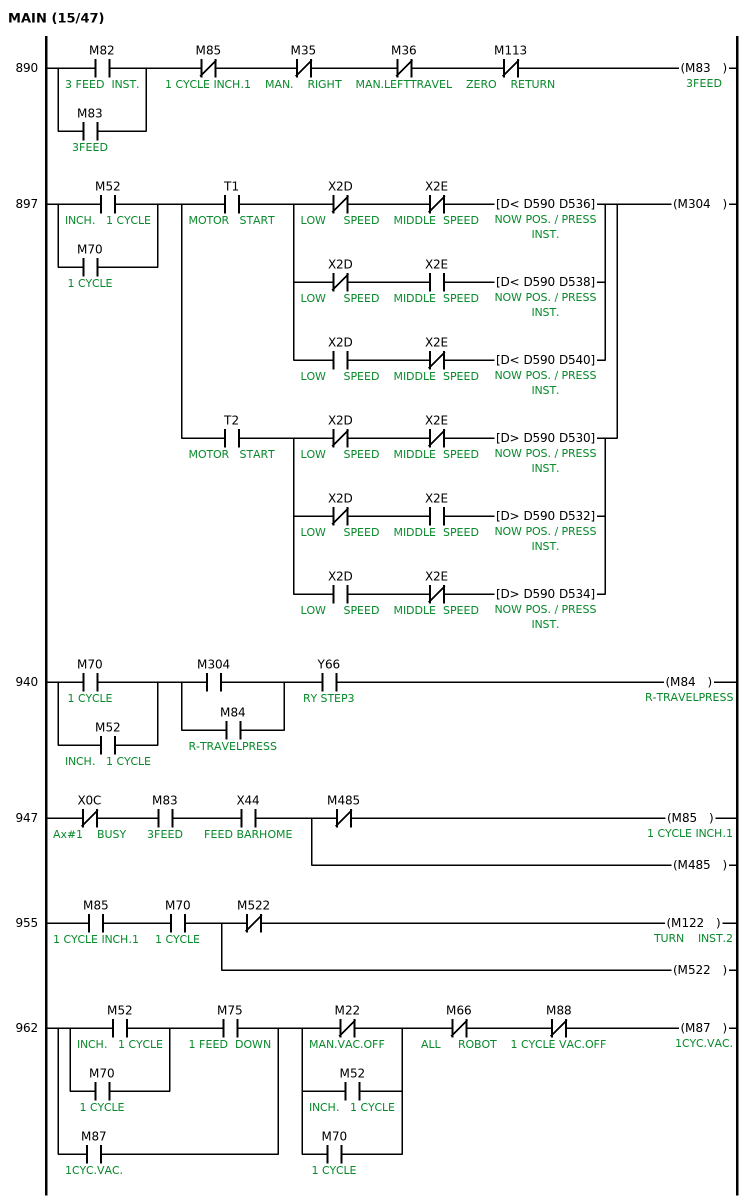
890   LD      M82  ; 3 FEED  INST.
      OR      M83  ; 3FEED
      ANI     M85  ; 1 CYCLE INCH.1
      ANI     M35  ; MAN.    RIGHT
      ANI     M36  ; MAN.LEFTTRAVEL
      ANI     M113  ; ZERO    RETURN
      OUT     M83  ; 3FEED
897   LD      M52  ; INCH.   1 CYCLE
      OR      M70  ; 1 CYCLE
      LD      T1  ; MOTOR   START
      LDI     X2D  ; LOW     SPEED
      ANI     X2E  ; MIDDLE  SPEED
      ANDD<   D590 D536  ; NOW POS. / PRESS   INST.
      LDI     X2D  ; LOW     SPEED
      AND     X2E  ; MIDDLE  SPEED
      ANDD<   D590 D538  ; NOW POS. / PRESS   INST.
      ORB
      LD      X2D  ; LOW     SPEED
      ANI     X2E  ; MIDDLE  SPEED
      ANDD<   D590 D540  ; NOW POS. / PRESS   INST.
      ORB
      ANB
      LD      T2  ; MOTOR   START
      LDI     X2D  ; LOW     SPEED
      ANI     X2E  ; MIDDLE  SPEED
      ANDD>   D590 D530  ; NOW POS. / PRESS   INST.
      LDI     X2D  ; LOW     SPEED
      AND     X2E  ; MIDDLE  SPEED
      ANDD>   D590 D532  ; NOW POS. / PRESS   INST.
      ORB
      LD      X2D  ; LOW     SPEED
      ANI     X2E  ; MIDDLE  SPEED
      ANDD>   D590 D534  ; NOW POS. / PRESS   INST.
      ORB
      ANB
      ORB
      ANB
      OUT     M304
940   LD      M70  ; 1 CYCLE
      OR      M52  ; INCH.   1 CYCLE
      LD      M304
      OR      M84  ; R-TRAVELPRESS
      ANB
      AND     Y66  ; RY STEP3
      OUT     M84  ; R-TRAVELPRESS
947   LDI     X0C  ; Ax#1    BUSY
      AND     M83  ; 3FEED
      AND     X44  ; FEED BARHOME
      MPS
      ANI     M485
      OUT     M85  ; 1 CYCLE INCH.1
      MPP
      OUT     M485
955   LD      M85  ; 1 CYCLE INCH.1
      AND     M70  ; 1 CYCLE
      MPS
      ANI     M522
      OUT     M122  ; TURN    INST.2
      MPP
      OUT     M522
962   LD      M52  ; INCH.   1 CYCLE
      OR      M70  ; 1 CYCLE
      AND     M75  ; 1 FEED  DOWN
      OR      M87  ; 1CYC.VAC.
      LDI     M22  ; MAN.VAC.OFF
      OR      M52  ; INCH.   1 CYCLE
      OR      M70  ; 1 CYCLE
      ANB
      ANI     M66  ; ALL     ROBOT
      ANI     M88  ; 1 CYCLE VAC.OFF
      OUT     M87  ; 1CYC.VAC.
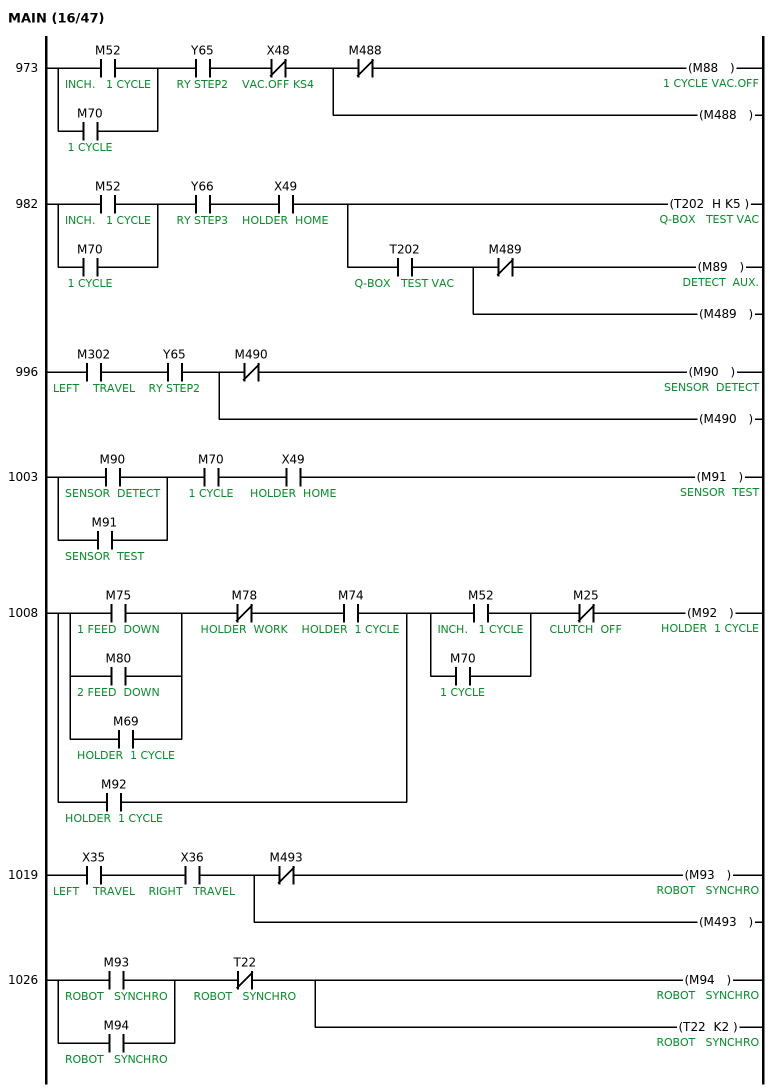
973   LD      M52  ; INCH.   1 CYCLE
      OR      M70  ; 1 CYCLE
      AND     Y65  ; RY STEP2
      ANI     X48  ; VAC.OFF KS4
      MPS
      ANI     M488
      OUT     M88  ; 1 CYCLE VAC.OFF
      MPP
      OUT     M488
982   LD      M52  ; INCH.   1 CYCLE
      OR      M70  ; 1 CYCLE
      AND     Y66  ; RY STEP3
      AND     X49  ; HOLDER  HOME
      OUTH    T202 K5  ; Q-BOX   TEST VAC
      AND     T202  ; Q-BOX   TEST VAC
      MPS
      ANI     M489
      OUT     M89  ; DETECT  AUX.
      MPP
      OUT     M489
996   LD      M302  ; LEFT    TRAVEL
      AND     Y65  ; RY STEP2
      MPS
      ANI     M490
      OUT     M90  ; SENSOR  DETECT
      MPP
      OUT     M490
1003  LD      M90  ; SENSOR  DETECT
      OR      M91  ; SENSOR  TEST
      AND     M70  ; 1 CYCLE
      AND     X49  ; HOLDER  HOME
      OUT     M91  ; SENSOR  TEST
1008  LD      M75  ; 1 FEED  DOWN
      OR      M80  ; 2 FEED  DOWN
      OR      M69  ; HOLDER  1 CYCLE
      ANI     M78  ; HOLDER  WORK
      AND     M74  ; HOLDER  1 CYCLE
      OR      M92  ; HOLDER  1 CYCLE
      LD      M52  ; INCH.   1 CYCLE
      OR      M70  ; 1 CYCLE
      ANB
      ANI     M25  ; CLUTCH  OFF
      OUT     M92  ; HOLDER  1 CYCLE
1019  LD      X35  ; LEFT    TRAVEL
      AND     X36  ; RIGHT   TRAVEL
      MPS
      ANI     M493
      OUT     M93  ; ROBOT   SYNCHRO
      MPP
      OUT     M493
1026  LD      M93  ; ROBOT   SYNCHRO
      OR      M94  ; ROBOT   SYNCHRO
      ANI     T22  ; ROBOT   SYNCHRO
      OUT     M94  ; ROBOT   SYNCHRO
      OUT     T22 K2  ; ROBOT   SYNCHRO
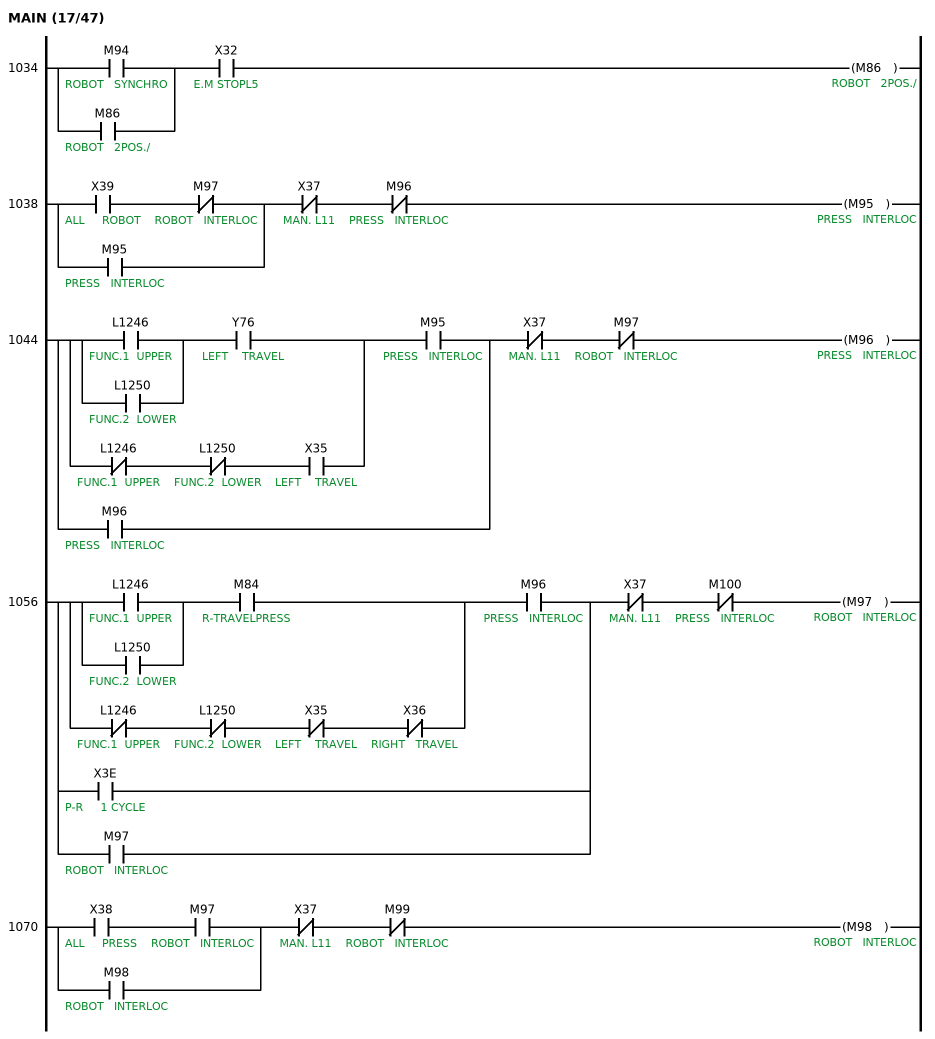
1034  LD      M94  ; ROBOT   SYNCHRO
      OR      M86  ; ROBOT   2POS./
      AND     X32  ; E.M STOPL5
      OUT     M86  ; ROBOT   2POS./
1038  LD      X39  ; ALL     ROBOT
      ANI     M97  ; ROBOT   INTERLOC
      OR      M95  ; PRESS   INTERLOC
      ANI     X37  ; MAN. L11
      ANI     M96  ; PRESS   INTERLOC
      OUT     M95  ; PRESS   INTERLOC
1044  LD      L1246  ; FUNC.1  UPPER
      OR      L1250  ; FUNC.2  LOWER
      AND     Y76  ; LEFT    TRAVEL
      LDI     L1246  ; FUNC.1  UPPER
      ANI     L1250  ; FUNC.2  LOWER
      AND     X35  ; LEFT    TRAVEL
      ORB
      AND     M95  ; PRESS   INTERLOC
      OR      M96  ; PRESS   INTERLOC
      ANI     X37  ; MAN. L11
      ANI     M97  ; ROBOT   INTERLOC
      OUT     M96  ; PRESS   INTERLOC
1056  LD      L1246  ; FUNC.1  UPPER
      OR      L1250  ; FUNC.2  LOWER
      AND     M84  ; R-TRAVELPRESS
      LDI     L1246  ; FUNC.1  UPPER
      ANI     L1250  ; FUNC.2  LOWER
      ANI     X35  ; LEFT    TRAVEL
      ANI     X36  ; RIGHT   TRAVEL
      ORB
      AND     M96  ; PRESS   INTERLOC
      OR      X3E  ; P-R     1 CYCLE
      OR      M97  ; ROBOT   INTERLOC
      ANI     X37  ; MAN. L11
      ANI     M100  ; PRESS   INTERLOC
      OUT     M97  ; ROBOT   INTERLOC
1070  LD      X38  ; ALL     PRESS
      AND     M97  ; ROBOT   INTERLOC
      OR      M98  ; ROBOT   INTERLOC
      ANI     X37  ; MAN. L11
      ANI     M99  ; ROBOT   INTERLOC
      OUT     M98  ; ROBOT   INTERLOC
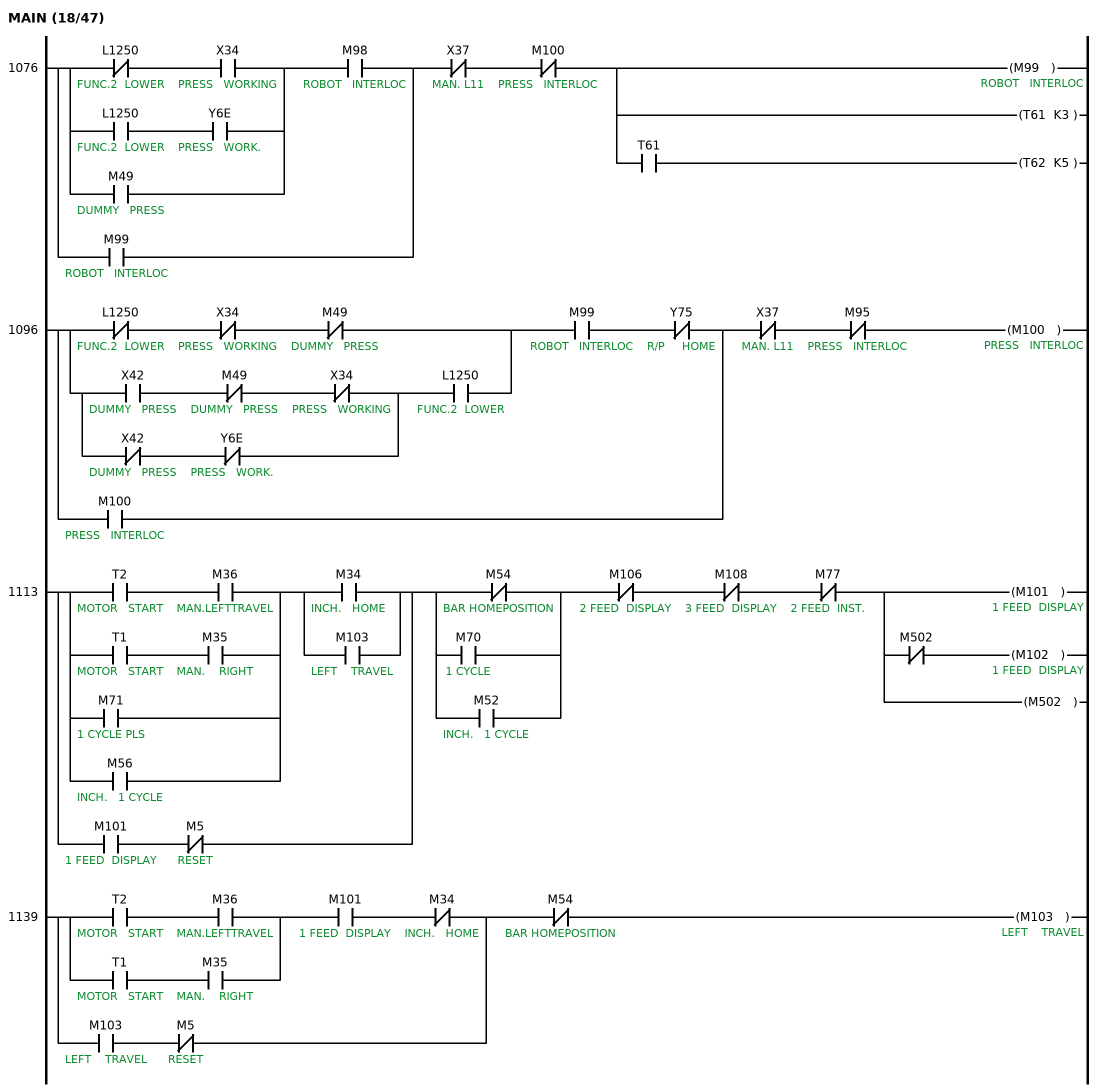
1076  LDI     L1250  ; FUNC.2  LOWER
      AND     X34  ; PRESS   WORKING
      LD      L1250  ; FUNC.2  LOWER
      AND     Y6E  ; PRESS   WORK.
      ORB
      OR      M49  ; DUMMY   PRESS
      AND     M98  ; ROBOT   INTERLOC
      OR      M99  ; ROBOT   INTERLOC
      ANI     X37  ; MAN. L11
      ANI     M100  ; PRESS   INTERLOC
      OUT     M99  ; ROBOT   INTERLOC
      OUT     T61 K3
      AND     T61
      OUT     T62 K5
1096  LDI     L1250  ; FUNC.2  LOWER
      ANI     X34  ; PRESS   WORKING
      ANI     M49  ; DUMMY   PRESS
      LD      X42  ; DUMMY   PRESS
      ANI     M49  ; DUMMY   PRESS
      ANI     X34  ; PRESS   WORKING
      LDI     X42  ; DUMMY   PRESS
      ANI     Y6E  ; PRESS   WORK.
      ORB
      AND     L1250  ; FUNC.2  LOWER
      ORB
      AND     M99  ; ROBOT   INTERLOC
      ANI     Y75  ; R/P     HOME
      OR      M100  ; PRESS   INTERLOC
      ANI     X37  ; MAN. L11
      ANI     M95  ; PRESS   INTERLOC
      OUT     M100  ; PRESS   INTERLOC
1113  LD      T2  ; MOTOR   START
      AND     M36  ; MAN.LEFTTRAVEL
      LD      T1  ; MOTOR   START
      AND     M35  ; MAN.    RIGHT
      ORB
      OR      M71  ; 1 CYCLE PLS
      OR      M56  ; INCH.   1 CYCLE
      LD      M34  ; INCH.   HOME
      OR      M103  ; LEFT    TRAVEL
      ANB
      LD      M101  ; 1 FEED  DISPLAY
      ANI     M5  ; RESET
      ORB
      LDI     M54  ; BAR HOMEPOSITION
      OR      M70  ; 1 CYCLE
      OR      M52  ; INCH.   1 CYCLE
      ANB
      ANI     M106  ; 2 FEED  DISPLAY
      ANI     M108  ; 3 FEED  DISPLAY
      ANI     M77  ; 2 FEED  INST.
      OUT     M101  ; 1 FEED  DISPLAY
      MPS
      ANI     M502
      OUT     M102  ; 1 FEED  DISPLAY
      MPP
      OUT     M502
1139  LD      T2  ; MOTOR   START
      AND     M36  ; MAN.LEFTTRAVEL
      LD      T1  ; MOTOR   START
      AND     M35  ; MAN.    RIGHT
      ORB
      AND     M101  ; 1 FEED  DISPLAY
      ANI     M34  ; INCH.   HOME
      LD      M103  ; LEFT    TRAVEL
      ANI     M5  ; RESET
      ORB
      ANI     M54  ; BAR HOMEPOSITION
      OUT     M103  ; LEFT    TRAVEL
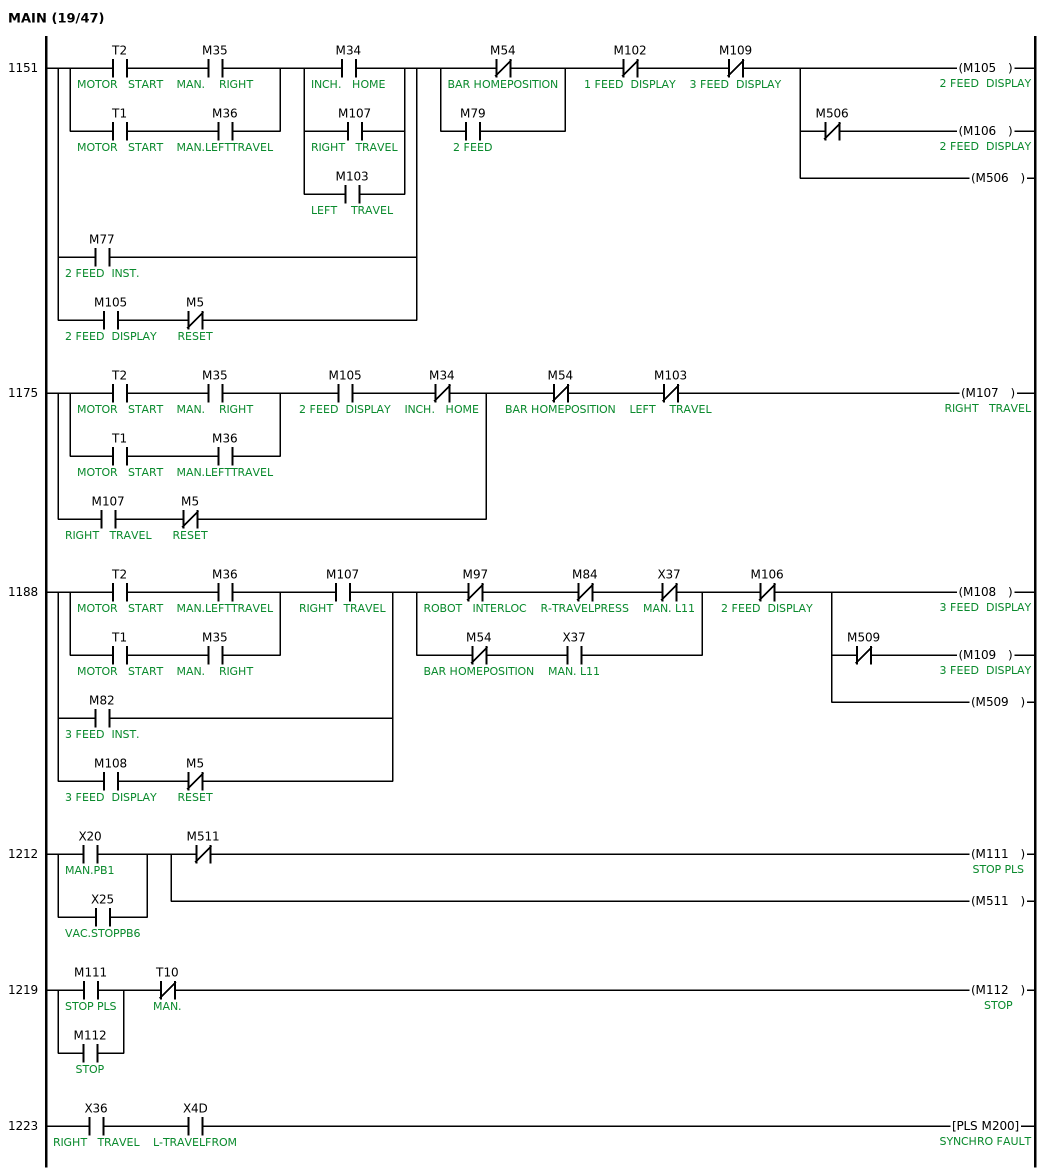
1151  LD      T2  ; MOTOR   START
      AND     M35  ; MAN.    RIGHT
      LD      T1  ; MOTOR   START
      AND     M36  ; MAN.LEFTTRAVEL
      ORB
      LD      M34  ; INCH.   HOME
      OR      M107  ; RIGHT   TRAVEL
      OR      M103  ; LEFT    TRAVEL
      ANB
      OR      M77  ; 2 FEED  INST.
      LD      M105  ; 2 FEED  DISPLAY
      ANI     M5  ; RESET
      ORB
      LDI     M54  ; BAR HOMEPOSITION
      OR      M79  ; 2 FEED
      ANB
      ANI     M102  ; 1 FEED  DISPLAY
      ANI     M109  ; 3 FEED  DISPLAY
      OUT     M105  ; 2 FEED  DISPLAY
      MPS
      ANI     M506
      OUT     M106  ; 2 FEED  DISPLAY
      MPP
      OUT     M506
1175  LD      T2  ; MOTOR   START
      AND     M35  ; MAN.    RIGHT
      LD      T1  ; MOTOR   START
      AND     M36  ; MAN.LEFTTRAVEL
      ORB
      AND     M105  ; 2 FEED  DISPLAY
      ANI     M34  ; INCH.   HOME
      LD      M107  ; RIGHT   TRAVEL
      ANI     M5  ; RESET
      ORB
      ANI     M54  ; BAR HOMEPOSITION
      ANI     M103  ; LEFT    TRAVEL
      OUT     M107  ; RIGHT   TRAVEL
1188  LD      T2  ; MOTOR   START
      AND     M36  ; MAN.LEFTTRAVEL
      LD      T1  ; MOTOR   START
      AND     M35  ; MAN.    RIGHT
      ORB
      AND     M107  ; RIGHT   TRAVEL
      OR      M82  ; 3 FEED  INST.
      LD      M108  ; 3 FEED  DISPLAY
      ANI     M5  ; RESET
      ORB
      LDI     M97  ; ROBOT   INTERLOC
      ANI     M84  ; R-TRAVELPRESS
      ANI     X37  ; MAN. L11
      LDI     M54  ; BAR HOMEPOSITION
      AND     X37  ; MAN. L11
      ORB
      ANB
      ANI     M106  ; 2 FEED  DISPLAY
      OUT     M108  ; 3 FEED  DISPLAY
      MPS
      ANI     M509
      OUT     M109  ; 3 FEED  DISPLAY
      MPP
      OUT     M509
1212  LD      X20  ; MAN.PB1
      OR      X25  ; VAC.STOPPB6
      MPS
      ANI     M511
      OUT     M111  ; STOP PLS
      MPP
      OUT     M511
1219  LD      M111  ; STOP PLS
      OR      M112  ; STOP
      ANI     T10  ; MAN.
      OUT     M112  ; STOP
1223  LD      X36  ; RIGHT   TRAVEL
      AND     X4D  ; L-TRAVELFROM
      PLS     M200  ; SYNCHRO FAULT
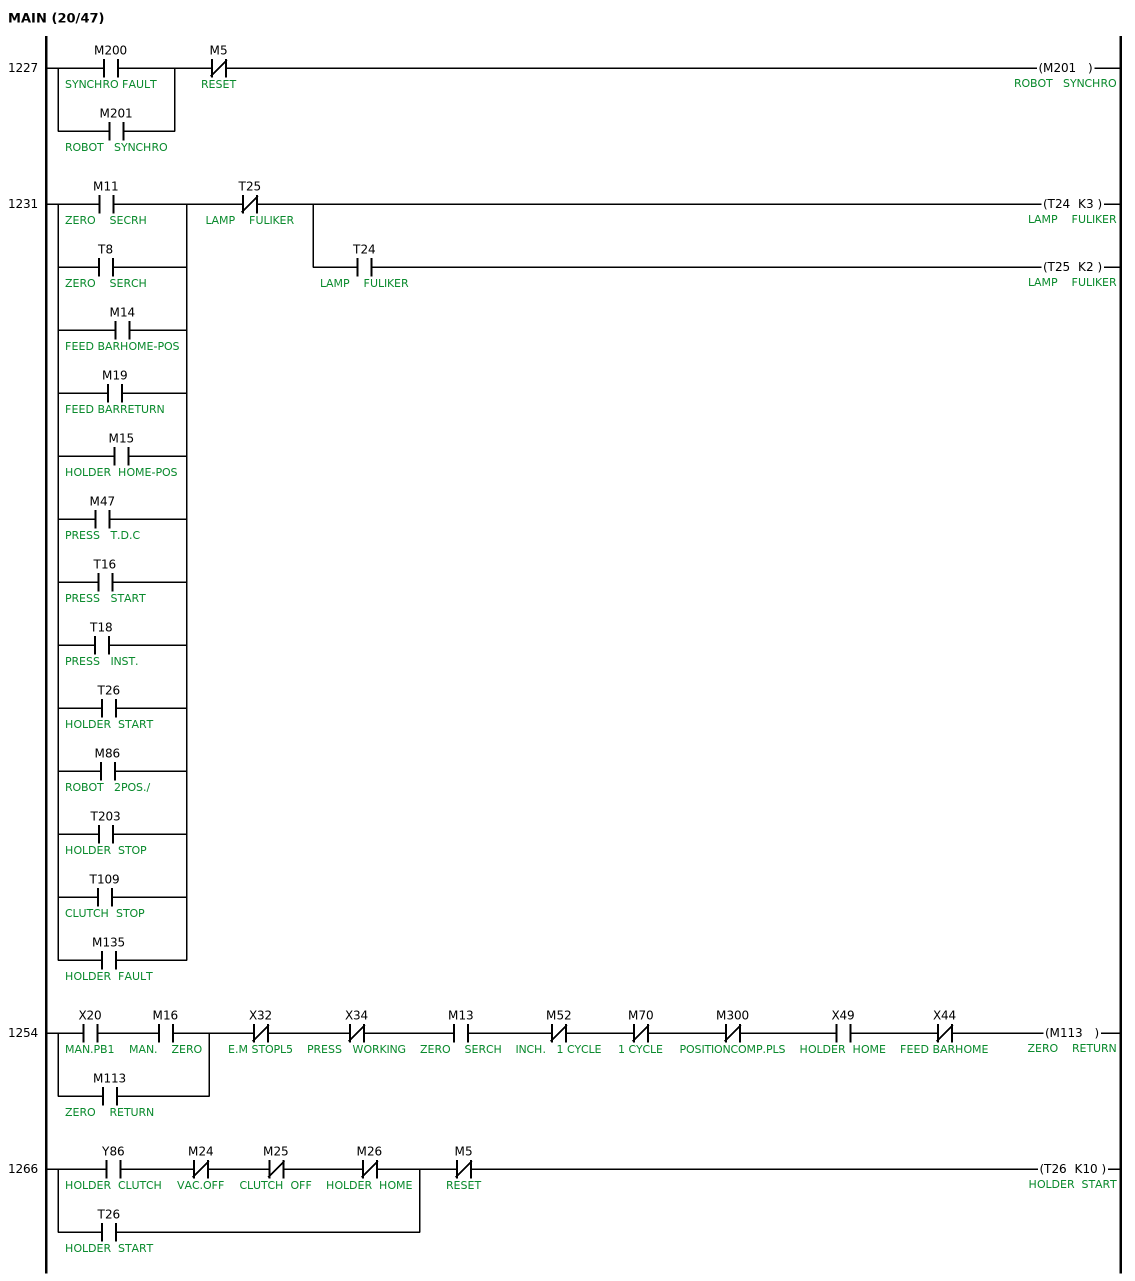
1227  LD      M200  ; SYNCHRO FAULT
      OR      M201  ; ROBOT   SYNCHRO
      ANI     M5  ; RESET
      OUT     M201  ; ROBOT   SYNCHRO
1231  LD      M11  ; ZERO    SECRH
      OR      T8  ; ZERO    SERCH
      OR      M14  ; FEED BARHOME-POS
      OR      M19  ; FEED BARRETURN
      OR      M15  ; HOLDER  HOME-POS
      OR      M47  ; PRESS   T.D.C
      OR      T16  ; PRESS   START
      OR      T18  ; PRESS   INST.
      OR      T26  ; HOLDER  START
      OR      M86  ; ROBOT   2POS./
      OR      T203  ; HOLDER  STOP
      OR      T109  ; CLUTCH  STOP
      OR      M135  ; HOLDER  FAULT
      ANI     T25  ; LAMP    FULIKER
      OUT     T24 K3  ; LAMP    FULIKER
      AND     T24  ; LAMP    FULIKER
      OUT     T25 K2  ; LAMP    FULIKER
1254  LD      X20  ; MAN.PB1
      AND     M16  ; MAN.    ZERO
      OR      M113  ; ZERO    RETURN
      ANI     X32  ; E.M STOPL5
      ANI     X34  ; PRESS   WORKING
      AND     M13  ; ZERO    SERCH
      ANI     M52  ; INCH.   1 CYCLE
      ANI     M70  ; 1 CYCLE
      ANI     M300  ; POSITIONCOMP.PLS
      AND     X49  ; HOLDER  HOME
      ANI     X44  ; FEED BARHOME
      OUT     M113  ; ZERO    RETURN
1266  LD      Y86  ; HOLDER  CLUTCH
      ANI     M24  ; VAC.OFF
      ANI     M25  ; CLUTCH  OFF
      ANI     M26  ; HOLDER  HOME
      OR      T26  ; HOLDER  START
      ANI     M5  ; RESET
      OUT     T26 K10  ; HOLDER  START
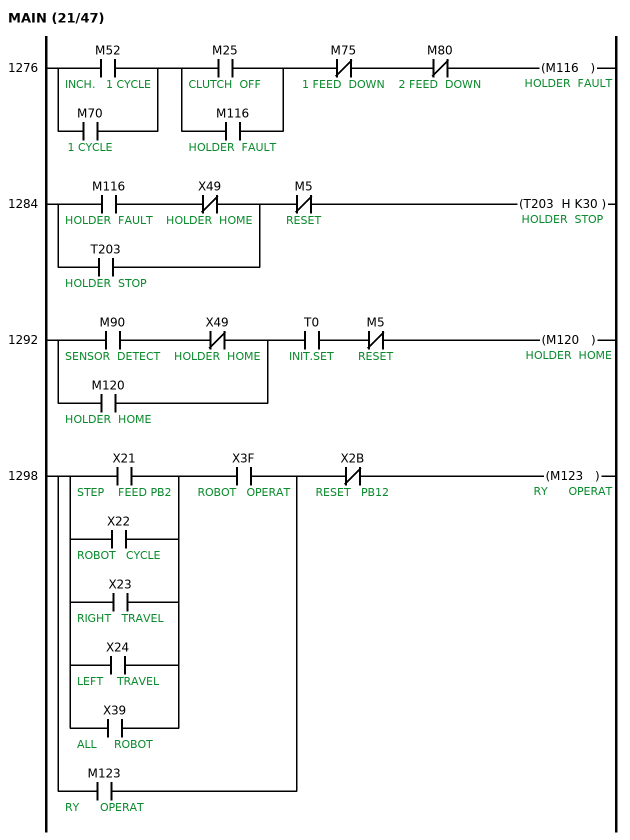
1276  LD      M52  ; INCH.   1 CYCLE
      OR      M70  ; 1 CYCLE
      LD      M25  ; CLUTCH  OFF
      OR      M116  ; HOLDER  FAULT
      ANB
      ANI     M75  ; 1 FEED  DOWN
      ANI     M80  ; 2 FEED  DOWN
      OUT     M116  ; HOLDER  FAULT
1284  LD      M116  ; HOLDER  FAULT
      ANI     X49  ; HOLDER  HOME
      OR      T203  ; HOLDER  STOP
      ANI     M5  ; RESET
      OUTH    T203 K30  ; HOLDER  STOP
1292  LD      M90  ; SENSOR  DETECT
      ANI     X49  ; HOLDER  HOME
      OR      M120  ; HOLDER  HOME
      AND     T0  ; INIT.SET
      ANI     M5  ; RESET
      OUT     M120  ; HOLDER  HOME
1298  LD      X21  ; STEP    FEED PB2
      OR      X22  ; ROBOT   CYCLE
      OR      X23  ; RIGHT   TRAVEL
      OR      X24  ; LEFT    TRAVEL
      OR      X39  ; ALL     ROBOT
      AND     X3F  ; ROBOT   OPERAT
      OR      M123  ; RY      OPERAT
      ANI     X2B  ; RESET   PB12
      OUT     M123  ; RY      OPERAT
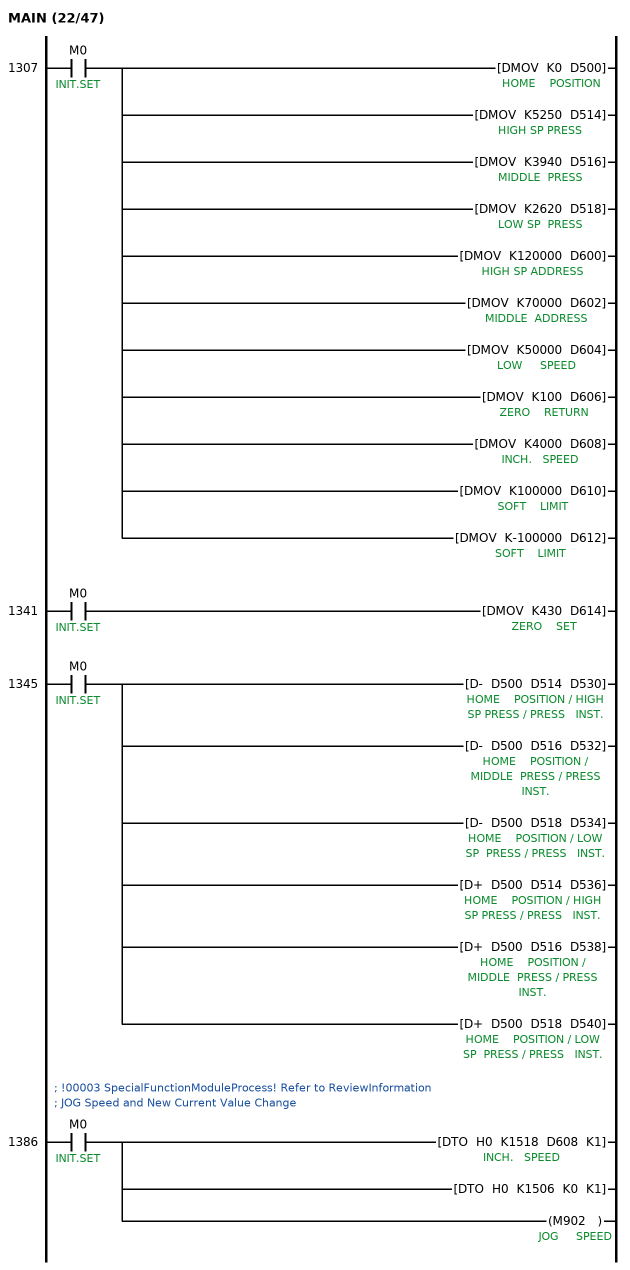
1307  LD      M0  ; INIT.SET
      DMOV    K0 D500  ; HOME    POSITION
      DMOV    K5250 D514  ; HIGH SP PRESS
      DMOV    K3940 D516  ; MIDDLE  PRESS
      DMOV    K2620 D518  ; LOW SP  PRESS
      DMOV    K120000 D600  ; HIGH SP ADDRESS
      DMOV    K70000 D602  ; MIDDLE  ADDRESS
      DMOV    K50000 D604  ; LOW     SPEED
      DMOV    K100 D606  ; ZERO    RETURN
      DMOV    K4000 D608  ; INCH.   SPEED
      DMOV    K100000 D610  ; SOFT    LIMIT
      DMOV    K-100000 D612  ; SOFT    LIMIT
1341  LD      M0  ; INIT.SET
      DMOV    K430 D614  ; ZERO    SET
1345  LD      M0  ; INIT.SET
      D-      D500 D514 D530
      D-      D500 D516 D532
      D-      D500 D518 D534
      D+      D500 D514 D536
      D+      D500 D516 D538
      D+      D500 D518 D540
; !00003 SpecialFunctionModuleProcess! Refer to ReviewInformation
; JOG Speed and New Current Value Change
1386  LD      M0  ; INIT.SET
      DTO     H0 K1518 D608 K1
      DTO     H0 K1506 K0 K1
      OUT     M902  ; JOG     SPEED
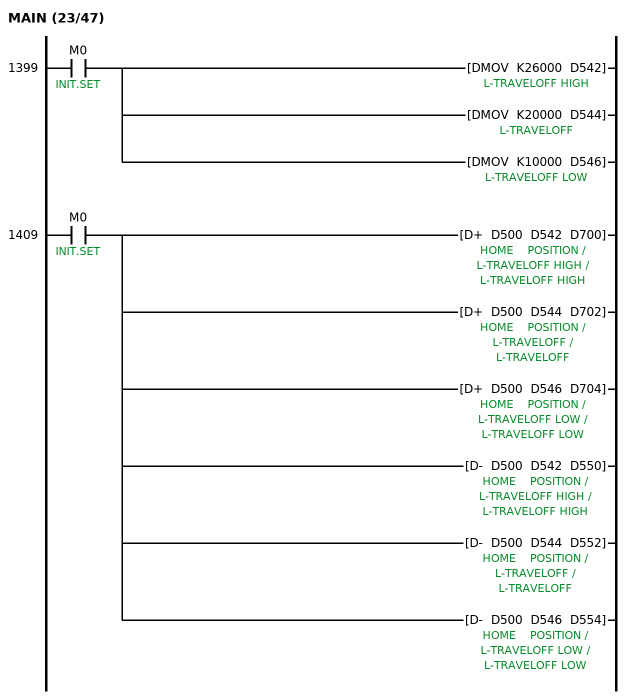
1399  LD      M0  ; INIT.SET
      DMOV    K26000 D542  ; L-TRAVELOFF HIGH
      DMOV    K20000 D544  ; L-TRAVELOFF
      DMOV    K10000 D546  ; L-TRAVELOFF LOW
1409  LD      M0  ; INIT.SET
      D+      D500 D542 D700
      D+      D500 D544 D702
      D+      D500 D546 D704
      D-      D500 D542 D550
      D-      D500 D544 D552
      D-      D500 D546 D554
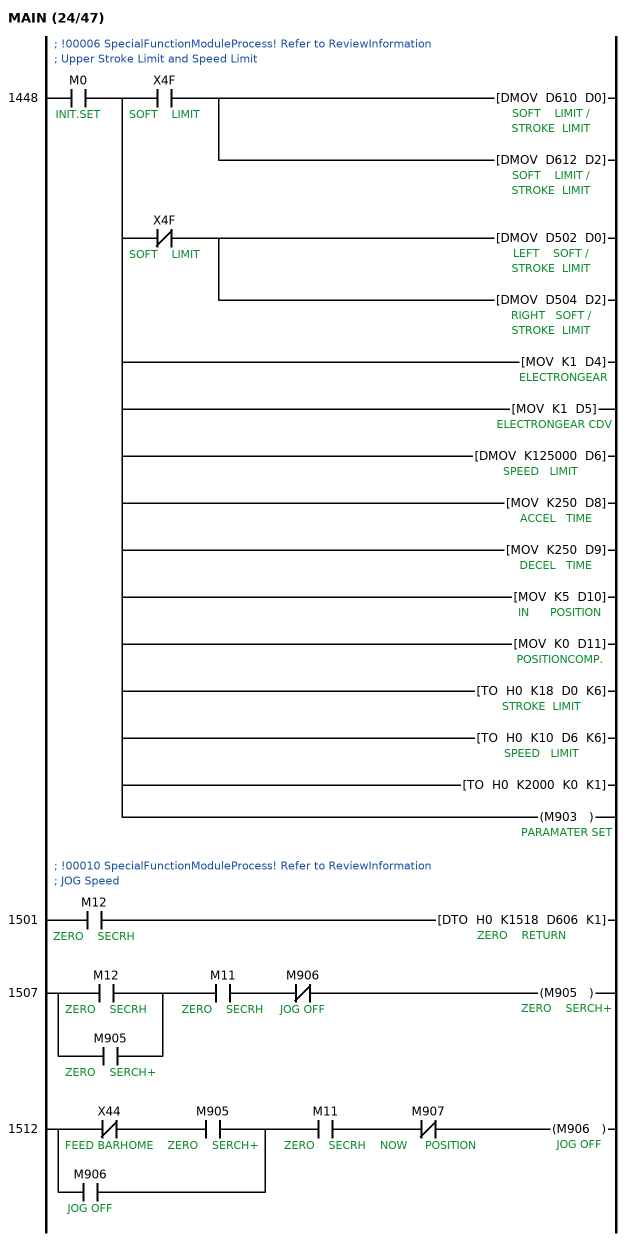
; !00006 SpecialFunctionModuleProcess! Refer to ReviewInformation
; Upper Stroke Limit and Speed Limit
1448  LD      M0  ; INIT.SET
      MPS
      AND     X4F  ; SOFT    LIMIT
      DMOV    D610 D0  ; STROKE  LIMIT
      DMOV    D612 D2  ; STROKE  LIMIT
      MRD
      ANI     X4F  ; SOFT    LIMIT
      DMOV    D502 D0  ; LEFT    SOFT
      DMOV    D504 D2  ; RIGHT   SOFT
      MPP
      MOV     K1 D4  ; ELECTRONGEAR
      MOV     K1 D5  ; ELECTRONGEAR CDV
      DMOV    K125000 D6  ; SPEED   LIMIT
      MOV     K250 D8  ; ACCEL   TIME
      MOV     K250 D9  ; DECEL   TIME
      MOV     K5 D10  ; IN      POSITION
      MOV     K0 D11  ; POSITIONCOMP.
      TO      H0 K18 D0 K6
      TO      H0 K10 D6 K6
      TO      H0 K2000 K0 K1
      OUT     M903  ; PARAMATER SET
; !00010 SpecialFunctionModuleProcess! Refer to ReviewInformation
; JOG Speed
1501  LD      M12  ; ZERO    SECRH
      DTO     H0 K1518 D606 K1
1507  LD      M12  ; ZERO    SECRH
      OR      M905  ; ZERO    SERCH+
      AND     M11  ; ZERO    SECRH
      ANI     M906  ; JOG OFF
      OUT     M905  ; ZERO    SERCH+
1512  LDI     X44  ; FEED BARHOME
      AND     M905  ; ZERO    SERCH+
      OR      M906  ; JOG OFF
      AND     M11  ; ZERO    SECRH
      ANI     M907  ; NOW     POSITION
      OUT     M906  ; JOG OFF
